Yaskawa INFORM job: DEMO_ROOF_UPPER_0625_3PAINT_16.JBI

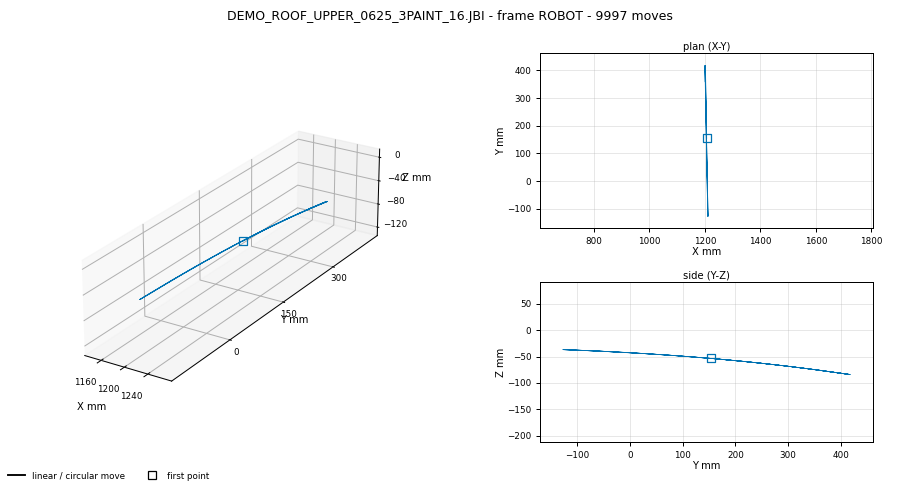
[picture p0: tool path of DEMO_ROOF_UPPER_0625_3PAINT_16.JBI in frame ROBOT, 9997 of 9997 moves have a stored position in this frame; points joined in program order, loops and branches not executed]
/JOB
//NAME DEMO_ROOF_UPPER_0625_3PAINT16
//POS
///NPOS 9997,0,0,0,0,0
///TOOL 0
///USER 0
///POSTYPE ROBOT
///RECTAN
///RCONF 1,0,0,0,0,0,0,0,0,0,0,0,0,0,0,0,0,0,0,0,0,0,0,0
C00000=1206.516,154.392,-53.585,-178.084,6.068,148.520
C00001=1206.512,154.641,-53.607,-178.082,6.070,148.519
C00002=1206.507,154.891,-53.628,-178.079,6.072,148.519
C00003=1206.502,155.139,-53.650,-178.077,6.072,148.518
C00004=1206.498,155.388,-53.670,-178.074,6.074,148.518
C00005=1206.493,155.637,-53.692,-178.071,6.076,148.517
C00006=1206.488,155.887,-53.713,-178.068,6.078,148.517
C00007=1206.483,156.135,-53.735,-178.066,6.078,148.517
C00008=1206.479,156.384,-53.757,-178.063,6.080,148.516
C00009=1206.473,156.633,-53.778,-178.060,6.082,148.516
C00010=1206.470,156.882,-53.799,-178.058,6.083,148.515
C00011=1206.465,157.131,-53.821,-178.056,6.085,148.515
C00012=1206.460,157.380,-53.842,-178.053,6.086,148.515
C00013=1206.456,157.630,-53.864,-178.050,6.087,148.514
C00014=1206.450,157.879,-53.885,-178.048,6.089,148.514
C00015=1206.445,158.127,-53.906,-178.045,6.091,148.513
C00016=1206.441,158.377,-53.928,-178.043,6.092,148.513
C00017=1206.436,158.625,-53.950,-178.040,6.093,148.512
C00018=1206.432,158.894,-53.973,-178.037,6.095,148.512
C00019=1206.426,159.164,-53.996,-178.034,6.097,148.511
C00020=1206.421,159.433,-54.019,-178.031,6.098,148.511
C00021=1206.416,159.702,-54.043,-178.028,6.100,148.510
C00022=1206.411,159.950,-54.065,-178.026,6.101,148.510
C00023=1206.407,160.200,-54.086,-178.023,6.102,148.509
C00024=1206.402,160.449,-54.108,-178.021,6.104,148.509
C00025=1206.397,160.698,-54.130,-178.018,6.106,148.509
C00026=1206.393,160.947,-54.152,-178.016,6.107,148.508
C00027=1206.388,161.196,-54.172,-178.013,6.109,148.508
C00028=1206.383,161.444,-54.194,-178.010,6.110,148.507
C00029=1206.379,161.694,-54.216,-178.008,6.111,148.507
C00030=1206.374,161.942,-54.237,-178.005,6.113,148.507
C00031=1206.370,162.192,-54.259,-178.002,6.115,148.506
C00032=1206.365,162.440,-54.281,-178.000,6.116,148.506
C00033=1206.360,162.690,-54.302,-177.997,6.117,148.505
C00034=1206.355,162.939,-54.325,-177.995,6.119,148.505
C00035=1206.350,163.188,-54.346,-177.992,6.121,148.505
C00036=1206.346,163.437,-54.368,-177.990,6.122,148.504
C00037=1206.341,163.686,-54.390,-177.987,6.123,148.504
C00038=1206.337,163.935,-54.412,-177.984,6.125,148.503
C00039=1206.332,164.184,-54.434,-177.981,6.127,148.503
C00040=1206.327,164.433,-54.456,-177.979,6.128,148.502
C00041=1206.323,164.682,-54.478,-177.977,6.130,148.502
C00042=1206.318,164.931,-54.499,-177.974,6.131,148.502
C00043=1206.314,165.180,-54.521,-177.971,6.133,148.501
C00044=1206.309,165.429,-54.543,-177.969,6.134,148.501
C00045=1206.304,165.678,-54.565,-177.966,6.136,148.500
C00046=1206.300,165.927,-54.587,-177.963,6.137,148.500
C00047=1206.295,166.176,-54.609,-177.961,6.139,148.500
C00048=1206.290,166.425,-54.631,-177.959,6.140,148.499
C00049=1206.285,166.674,-54.653,-177.955,6.142,148.499
C00050=1206.281,166.923,-54.675,-177.953,6.143,148.498
C00051=1206.276,167.171,-54.696,-177.950,6.145,148.498
C00052=1206.271,167.421,-54.718,-177.948,6.146,148.498
C00053=1206.267,167.669,-54.740,-177.945,6.148,148.497
C00054=1206.262,167.919,-54.762,-177.943,6.150,148.497
C00055=1206.257,168.168,-54.784,-177.939,6.151,148.496
C00056=1206.252,168.417,-54.807,-177.937,6.152,148.496
C00057=1206.248,168.666,-54.828,-177.935,6.154,148.495
C00058=1206.244,168.914,-54.851,-177.932,6.156,148.495
C00059=1206.239,169.163,-54.873,-177.929,6.158,148.495
C00060=1206.234,169.413,-54.895,-177.927,6.159,148.494
C00061=1206.229,169.661,-54.917,-177.924,6.160,148.494
C00062=1206.225,169.911,-54.939,-177.921,6.162,148.493
C00063=1206.220,170.160,-54.961,-177.919,6.164,148.493
C00064=1206.215,170.408,-54.984,-177.916,6.166,148.493
C00065=1206.211,170.658,-55.006,-177.914,6.166,148.492
C00066=1206.206,170.906,-55.028,-177.911,6.168,148.492
C00067=1206.202,171.156,-55.050,-177.909,6.170,148.492
C00068=1206.196,171.405,-55.072,-177.906,6.172,148.491
C00069=1206.192,171.653,-55.095,-177.903,6.173,148.491
C00070=1206.187,171.902,-55.117,-177.901,6.174,148.490
C00071=1206.183,172.151,-55.139,-177.898,6.176,148.490
C00072=1206.178,172.401,-55.161,-177.895,6.178,148.489
C00073=1206.173,172.649,-55.184,-177.893,6.180,148.489
C00074=1206.169,172.898,-55.206,-177.891,6.181,148.489
C00075=1206.163,173.147,-55.228,-177.888,6.182,148.488
C00076=1206.159,173.396,-55.251,-177.885,6.184,148.488
C00077=1206.155,173.645,-55.272,-177.882,6.186,148.487
C00078=1206.150,173.894,-55.295,-177.880,6.188,148.487
C00079=1206.146,174.143,-55.318,-177.877,6.189,148.487
C00080=1206.141,174.392,-55.340,-177.875,6.190,148.486
C00081=1206.136,174.641,-55.362,-177.872,6.192,148.486
C00082=1206.132,174.890,-55.385,-177.869,6.194,148.486
C00083=1206.127,175.139,-55.407,-177.866,6.196,148.485
C00084=1206.122,175.388,-55.430,-177.864,6.197,148.485
C00085=1206.117,175.636,-55.452,-177.862,6.198,148.484
C00086=1206.112,175.886,-55.474,-177.859,6.200,148.484
C00087=1206.108,176.135,-55.497,-177.856,6.202,148.484
C00088=1206.104,176.383,-55.519,-177.854,6.204,148.483
C00089=1206.099,176.632,-55.542,-177.851,6.205,148.483
C00090=1206.095,176.882,-55.564,-177.849,6.207,148.482
C00091=1206.089,177.130,-55.587,-177.846,6.208,148.482
C00092=1206.085,177.379,-55.609,-177.843,6.210,148.482
C00093=1206.081,177.628,-55.632,-177.840,6.212,148.481
C00094=1206.075,177.877,-55.654,-177.838,6.213,148.481
C00095=1206.071,178.126,-55.677,-177.836,6.214,148.480
C00096=1206.066,178.375,-55.700,-177.833,6.216,148.480
C00097=1206.062,178.623,-55.722,-177.830,6.218,148.480
C00098=1206.057,178.873,-55.745,-177.828,6.220,148.479
C00099=1206.053,179.122,-55.767,-177.825,6.222,148.479
C00100=1206.047,179.371,-55.790,-177.823,6.223,148.479
C00101=1206.043,179.620,-55.813,-177.820,6.224,148.478
C00102=1206.039,179.869,-55.836,-177.817,6.226,148.478
C00103=1206.034,180.118,-55.858,-177.814,6.228,148.477
C00104=1206.029,180.366,-55.881,-177.812,6.230,148.477
C00105=1206.025,180.616,-55.903,-177.809,6.231,148.477
C00106=1206.020,180.865,-55.926,-177.806,6.233,148.476
C00107=1206.016,181.113,-55.949,-177.804,6.234,148.476
C00108=1206.011,181.362,-55.971,-177.802,6.236,148.476
C00109=1206.007,181.611,-55.994,-177.799,6.238,148.475
C00110=1206.002,181.860,-56.017,-177.796,6.240,148.475
C00111=1205.996,182.109,-56.040,-177.794,6.241,148.474
C00112=1205.992,182.358,-56.063,-177.791,6.243,148.474
C00113=1205.988,182.607,-56.086,-177.789,6.244,148.474
C00114=1205.984,182.855,-56.109,-177.786,6.246,148.473
C00115=1205.978,183.104,-56.131,-177.784,6.248,148.473
C00116=1205.973,183.353,-56.154,-177.780,6.249,148.472
C00117=1205.969,183.602,-56.177,-177.778,6.251,148.472
C00118=1205.964,183.852,-56.200,-177.775,6.253,148.472
C00119=1205.960,184.101,-56.222,-177.772,6.255,148.471
C00120=1205.955,184.349,-56.245,-177.770,6.256,148.471
C00121=1205.950,184.598,-56.269,-177.768,6.258,148.471
C00122=1205.946,184.867,-56.293,-177.765,6.259,148.470
C00123=1205.941,185.137,-56.318,-177.762,6.262,148.470
C00124=1205.935,185.407,-56.343,-177.759,6.264,148.470
C00125=1205.931,185.676,-56.368,-177.756,6.265,148.469
C00126=1205.926,185.925,-56.391,-177.753,6.267,148.469
C00127=1205.921,186.174,-56.414,-177.751,6.269,148.468
C00128=1205.917,186.423,-56.437,-177.749,6.270,148.468
C00129=1205.913,186.672,-56.461,-177.746,6.272,148.468
C00130=1205.907,186.920,-56.484,-177.743,6.274,148.467
C00131=1205.903,187.170,-56.506,-177.741,6.275,148.467
C00132=1205.898,187.419,-56.529,-177.738,6.277,148.467
C00133=1205.894,187.668,-56.552,-177.735,6.279,148.466
C00134=1205.889,187.917,-56.576,-177.733,6.281,148.466
C00135=1205.885,188.166,-56.598,-177.730,6.283,148.465
C00136=1205.880,188.414,-56.621,-177.727,6.284,148.465
C00137=1205.875,188.663,-56.645,-177.725,6.285,148.465
C00138=1205.870,188.912,-56.668,-177.723,6.287,148.464
C00139=1205.866,189.161,-56.691,-177.720,6.289,148.464
C00140=1205.862,189.410,-56.714,-177.717,6.291,148.464
C00141=1205.857,189.659,-56.738,-177.715,6.293,148.463
C00142=1205.852,189.908,-56.761,-177.712,6.295,148.463
C00143=1205.847,190.157,-56.784,-177.709,6.296,148.463
C00144=1205.844,190.406,-56.807,-177.707,6.298,148.462
C00145=1205.838,190.654,-56.830,-177.704,6.300,148.462
C00146=1205.834,190.903,-56.854,-177.701,6.302,148.462
C00147=1205.829,191.152,-56.877,-177.699,6.303,148.461
C00148=1205.824,191.401,-56.900,-177.697,6.305,148.461
C00149=1205.820,191.649,-56.924,-177.694,6.306,148.460
C00150=1205.816,191.898,-56.947,-177.691,6.308,148.460
C00151=1205.811,192.147,-56.970,-177.689,6.310,148.460
C00152=1205.806,192.396,-56.994,-177.686,6.312,148.459
C00153=1205.802,192.645,-57.017,-177.683,6.314,148.459
C00154=1205.797,192.894,-57.040,-177.681,6.316,148.459
C00155=1205.792,193.143,-57.064,-177.678,6.317,148.458
C00156=1205.788,193.392,-57.088,-177.675,6.319,148.458
C00157=1205.783,193.641,-57.111,-177.673,6.321,148.458
C00158=1205.778,193.890,-57.135,-177.670,6.323,148.457
C00159=1205.774,194.139,-57.157,-177.667,6.325,148.457
C00160=1205.769,194.387,-57.180,-177.665,6.326,148.457
C00161=1205.765,194.635,-57.204,-177.663,6.327,148.456
C00162=1205.760,194.884,-57.228,-177.660,6.329,148.456
C00163=1205.755,195.133,-57.251,-177.657,6.331,148.456
C00164=1205.751,195.382,-57.275,-177.655,6.333,148.455
C00165=1205.746,195.631,-57.299,-177.652,6.335,148.455
C00166=1205.742,195.880,-57.322,-177.649,6.337,148.455
C00167=1205.737,196.129,-57.345,-177.647,6.338,148.454
C00168=1205.732,196.378,-57.369,-177.644,6.340,148.454
C00169=1205.728,196.626,-57.393,-177.641,6.342,148.454
C00170=1205.723,196.875,-57.416,-177.639,6.344,148.453
C00171=1205.718,197.124,-57.439,-177.636,6.346,148.453
C00172=1205.714,197.373,-57.464,-177.634,6.347,148.452
C00173=1205.710,197.623,-57.487,-177.631,6.349,148.452
C00174=1205.706,197.871,-57.511,-177.628,6.351,148.452
C00175=1205.701,198.120,-57.535,-177.626,6.353,148.451
C00176=1205.696,198.369,-57.558,-177.623,6.355,148.451
C00177=1205.692,198.617,-57.582,-177.620,6.357,148.451
C00178=1205.687,198.866,-57.606,-177.618,6.358,148.450
C00179=1205.683,199.115,-57.630,-177.615,6.360,148.450
C00180=1205.677,199.364,-57.654,-177.613,6.361,148.450
C00181=1205.672,199.613,-57.677,-177.610,6.363,148.449
C00182=1205.668,199.862,-57.701,-177.608,6.365,148.449
C00183=1205.663,200.111,-57.724,-177.605,6.367,148.449
C00184=1205.659,200.359,-57.748,-177.602,6.369,148.448
C00185=1205.654,200.608,-57.772,-177.600,6.370,148.448
C00186=1205.650,200.857,-57.796,-177.597,6.372,148.448
C00187=1205.645,201.106,-57.819,-177.595,6.374,148.448
C00188=1205.641,201.355,-57.844,-177.592,6.376,148.447
C00189=1205.636,201.604,-57.868,-177.590,6.378,148.447
C00190=1205.632,201.852,-57.892,-177.587,6.380,148.446
C00191=1205.627,202.101,-57.916,-177.584,6.382,148.446
C00192=1205.622,202.350,-57.939,-177.582,6.383,148.446
C00193=1205.618,202.598,-57.963,-177.579,6.385,148.445
C00194=1205.613,202.847,-57.987,-177.576,6.387,148.445
C00195=1205.608,203.096,-58.011,-177.574,6.389,148.445
C00196=1205.604,203.345,-58.036,-177.571,6.391,148.444
C00197=1205.600,203.594,-58.059,-177.568,6.393,148.444
C00198=1205.595,203.843,-58.083,-177.566,6.394,148.444
C00199=1205.591,204.092,-58.106,-177.563,6.396,148.443
C00200=1205.586,204.340,-58.131,-177.560,6.398,148.443
C00201=1205.581,204.589,-58.155,-177.558,6.400,148.443
C00202=1205.576,204.838,-58.179,-177.556,6.402,148.443
C00203=1205.573,205.087,-58.203,-177.553,6.404,148.442
C00204=1205.568,205.335,-58.227,-177.550,6.406,148.442
C00205=1205.563,205.584,-58.252,-177.548,6.408,148.442
C00206=1205.558,205.833,-58.275,-177.545,6.409,148.441
C00207=1205.554,206.081,-58.299,-177.542,6.411,148.441
C00208=1205.550,206.331,-58.324,-177.540,6.413,148.441
C00209=1205.545,206.580,-58.348,-177.537,6.415,148.440
C00210=1205.540,206.828,-58.372,-177.534,6.417,148.440
C00211=1205.536,207.077,-58.396,-177.532,6.419,148.440
C00212=1205.531,207.325,-58.420,-177.529,6.420,148.439
C00213=1205.527,207.575,-58.445,-177.527,6.423,148.439
C00214=1205.522,207.824,-58.468,-177.524,6.424,148.439
C00215=1205.517,208.072,-58.493,-177.522,6.426,148.438
C00216=1205.513,208.321,-58.517,-177.519,6.428,148.438
C00217=1205.508,208.569,-58.541,-177.516,6.430,148.438
C00218=1205.504,208.819,-58.566,-177.514,6.432,148.437
C00219=1205.500,209.067,-58.590,-177.511,6.433,148.437
C00220=1205.494,209.316,-58.615,-177.508,6.436,148.437
C00221=1205.490,209.565,-58.638,-177.505,6.438,148.436
C00222=1205.486,209.814,-58.663,-177.503,6.440,148.436
C00223=1205.481,210.063,-58.687,-177.500,6.442,148.436
C00224=1205.476,210.311,-58.711,-177.498,6.444,148.436
C00225=1205.471,210.560,-58.736,-177.495,6.446,148.435
C00226=1205.467,210.830,-58.762,-177.492,6.447,148.435
C00227=1205.462,211.100,-58.789,-177.490,6.449,148.435
C00228=1205.457,211.371,-58.815,-177.487,6.452,148.434
C00229=1205.452,211.641,-58.842,-177.484,6.454,148.434
C00230=1205.448,211.891,-58.866,-177.481,6.456,148.434
C00231=1205.443,212.139,-58.891,-177.479,6.457,148.433
C00232=1205.438,212.388,-58.915,-177.476,6.459,148.433
C00233=1205.434,212.637,-58.940,-177.473,6.461,148.433
C00234=1205.429,212.886,-58.964,-177.471,6.463,148.432
C00235=1205.424,213.134,-58.989,-177.468,6.465,148.432
C00236=1205.421,213.383,-59.013,-177.466,6.467,148.432
C00237=1205.415,213.632,-59.038,-177.463,6.469,148.432
C00238=1205.411,213.880,-59.063,-177.461,6.471,148.431
C00239=1205.406,214.129,-59.087,-177.457,6.473,148.431
C00240=1205.402,214.378,-59.112,-177.455,6.475,148.431
C00241=1205.397,214.626,-59.137,-177.452,6.477,148.430
C00242=1205.393,214.876,-59.161,-177.450,6.479,148.430
C00243=1205.388,215.124,-59.186,-177.447,6.481,148.430
C00244=1205.384,215.373,-59.210,-177.445,6.483,148.429
C00245=1205.379,215.622,-59.235,-177.442,6.485,148.429
C00246=1205.375,215.870,-59.260,-177.439,6.486,148.429
C00247=1205.370,216.119,-59.284,-177.437,6.488,148.428
C00248=1205.366,216.368,-59.309,-177.434,6.490,148.428
C00249=1205.361,216.616,-59.333,-177.432,6.492,148.428
C00250=1205.356,216.865,-59.358,-177.429,6.494,148.428
C00251=1205.353,217.114,-59.383,-177.427,6.496,148.427
C00252=1205.348,217.362,-59.408,-177.424,6.499,148.427
C00253=1205.343,217.612,-59.433,-177.421,6.500,148.427
C00254=1205.339,217.860,-59.457,-177.418,6.502,148.426
C00255=1205.334,218.109,-59.483,-177.416,6.504,148.426
C00256=1205.329,218.358,-59.507,-177.413,6.506,148.426
C00257=1205.325,218.606,-59.531,-177.411,6.508,148.426
C00258=1205.321,218.855,-59.557,-177.408,6.510,148.425
C00259=1205.316,219.103,-59.581,-177.406,6.512,148.425
C00260=1205.312,219.353,-59.606,-177.403,6.514,148.425
C00261=1205.307,219.601,-59.632,-177.401,6.516,148.424
C00262=1205.303,219.850,-59.656,-177.398,6.518,148.424
C00263=1205.298,220.099,-59.681,-177.395,6.520,148.424
C00264=1205.293,220.347,-59.706,-177.392,6.522,148.424
C00265=1205.289,220.596,-59.731,-177.390,6.524,148.423
C00266=1205.284,220.845,-59.755,-177.387,6.526,148.423
C00267=1205.280,221.094,-59.781,-177.385,6.528,148.423
C00268=1205.275,221.342,-59.806,-177.382,6.530,148.422
C00269=1205.271,221.591,-59.831,-177.380,6.532,148.422
C00270=1205.266,221.839,-59.856,-177.377,6.533,148.422
C00271=1205.262,222.088,-59.881,-177.375,6.536,148.422
C00272=1205.257,222.337,-59.906,-177.372,6.537,148.421
C00273=1205.253,222.585,-59.931,-177.369,6.540,148.421
C00274=1205.248,222.834,-59.956,-177.366,6.542,148.421
C00275=1205.244,223.083,-59.982,-177.364,6.544,148.420
C00276=1205.239,223.332,-60.006,-177.361,6.546,148.420
C00277=1205.235,223.581,-60.032,-177.359,6.548,148.420
C00278=1205.230,223.829,-60.056,-177.356,6.550,148.420
C00279=1205.226,224.078,-60.082,-177.354,6.551,148.419
C00280=1205.221,224.326,-60.106,-177.351,6.554,148.419
C00281=1205.217,224.575,-60.132,-177.348,6.556,148.419
C00282=1205.212,224.824,-60.157,-177.346,6.558,148.419
C00283=1205.207,225.073,-60.183,-177.343,6.560,148.418
C00284=1205.203,225.321,-60.207,-177.341,6.562,148.418
C00285=1205.199,225.570,-60.232,-177.338,6.564,148.418
C00286=1205.194,225.819,-60.258,-177.335,6.566,148.417
C00287=1205.189,226.068,-60.283,-177.333,6.568,148.417
C00288=1205.185,226.316,-60.309,-177.330,6.569,148.417
C00289=1205.180,226.564,-60.334,-177.328,6.572,148.417
C00290=1205.176,226.814,-60.359,-177.325,6.574,148.416
C00291=1205.171,227.062,-60.384,-177.322,6.576,148.416
C00292=1205.167,227.311,-60.410,-177.320,6.578,148.416
C00293=1205.163,227.559,-60.435,-177.317,6.580,148.416
C00294=1205.158,227.808,-60.460,-177.315,6.582,148.415
C00295=1205.154,228.057,-60.486,-177.312,6.584,148.415
C00296=1205.149,228.305,-60.511,-177.310,6.586,148.415
C00297=1205.145,228.554,-60.536,-177.307,6.589,148.415
C00298=1205.140,228.803,-60.562,-177.304,6.591,148.414
C00299=1205.135,229.051,-60.587,-177.302,6.592,148.414
C00300=1205.131,229.300,-60.613,-177.299,6.595,148.414
C00301=1205.126,229.548,-60.638,-177.297,6.596,148.414
C00302=1205.122,229.798,-60.663,-177.294,6.598,148.413
C00303=1205.118,230.046,-60.689,-177.291,6.600,148.413
C00304=1205.113,230.294,-60.715,-177.289,6.603,148.413
C00305=1205.109,230.543,-60.740,-177.286,6.605,148.413
C00306=1205.104,230.792,-60.766,-177.283,6.607,148.412
C00307=1205.100,231.040,-60.791,-177.281,6.609,148.412
C00308=1205.095,231.290,-60.817,-177.279,6.611,148.412
C00309=1205.091,231.538,-60.842,-177.276,6.613,148.411
C00310=1205.086,231.787,-60.868,-177.273,6.614,148.411
C00311=1205.082,232.035,-60.893,-177.271,6.617,148.411
C00312=1205.078,232.284,-60.919,-177.268,6.619,148.411
C00313=1205.073,232.532,-60.945,-177.265,6.621,148.410
C00314=1205.068,232.781,-60.971,-177.263,6.623,148.410
C00315=1205.064,233.030,-60.997,-177.261,6.625,148.410
C00316=1205.059,233.278,-61.022,-177.258,6.627,148.410
C00317=1205.054,233.527,-61.048,-177.255,6.630,148.410
C00318=1205.050,233.776,-61.074,-177.253,6.632,148.409
C00319=1205.045,234.024,-61.099,-177.250,6.634,148.409
C00320=1205.041,234.273,-61.125,-177.247,6.636,148.409
C00321=1205.037,234.522,-61.150,-177.245,6.638,148.409
C00322=1205.033,234.770,-61.176,-177.243,6.640,148.408
C00323=1205.027,235.019,-61.202,-177.239,6.642,148.408
C00324=1205.023,235.268,-61.228,-177.237,6.644,148.408
C00325=1205.019,235.516,-61.254,-177.235,6.646,148.407
C00326=1205.014,235.765,-61.279,-177.232,6.648,148.407
C00327=1205.010,236.013,-61.305,-177.230,6.650,148.407
C00328=1205.005,236.262,-61.331,-177.227,6.653,148.407
C00329=1205.000,236.511,-61.357,-177.224,6.655,148.406
C00330=1204.995,236.782,-61.385,-177.222,6.657,148.406
C00331=1204.991,237.054,-61.413,-177.219,6.660,148.406
C00332=1204.986,237.325,-61.442,-177.216,6.661,148.406
C00333=1204.981,237.596,-61.470,-177.213,6.664,148.405
C00334=1204.977,237.845,-61.495,-177.211,6.666,148.405
C00335=1204.972,238.094,-61.522,-177.208,6.668,148.405
C00336=1204.968,238.342,-61.548,-177.205,6.670,148.405
C00337=1204.963,238.590,-61.574,-177.203,6.672,148.405
C00338=1204.959,238.839,-61.599,-177.200,6.675,148.404
C00339=1204.954,239.088,-61.626,-177.197,6.677,148.404
C00340=1204.950,239.337,-61.652,-177.195,6.679,148.404
C00341=1204.946,239.585,-61.678,-177.193,6.681,148.404
C00342=1204.940,239.834,-61.704,-177.190,6.683,148.403
C00343=1204.936,240.083,-61.730,-177.187,6.686,148.403
C00344=1204.932,240.331,-61.756,-177.185,6.687,148.403
C00345=1204.928,240.580,-61.782,-177.182,6.689,148.403
C00346=1204.923,240.829,-61.808,-177.180,6.691,148.403
C00347=1204.919,241.077,-61.834,-177.177,6.693,148.402
C00348=1204.914,241.325,-61.860,-177.175,6.696,148.402
C00349=1204.909,241.574,-61.886,-177.172,6.698,148.402
C00350=1204.905,241.822,-61.913,-177.169,6.700,148.402
C00351=1204.900,242.071,-61.939,-177.167,6.702,148.401
C00352=1204.896,242.320,-61.965,-177.164,6.705,148.401
C00353=1204.892,242.568,-61.992,-177.162,6.707,148.401
C00354=1204.887,242.817,-62.018,-177.159,6.709,148.401
C00355=1204.883,243.066,-62.044,-177.157,6.711,148.400
C00356=1204.879,243.314,-62.070,-177.154,6.713,148.400
C00357=1204.874,243.563,-62.096,-177.151,6.716,148.400
C00358=1204.870,243.811,-62.123,-177.149,6.717,148.400
C00359=1204.865,244.060,-62.149,-177.146,6.720,148.400
C00360=1204.861,244.308,-62.175,-177.144,6.721,148.399
C00361=1204.856,244.557,-62.202,-177.141,6.724,148.399
C00362=1204.852,244.806,-62.228,-177.138,6.726,148.399
C00363=1204.848,245.054,-62.254,-177.136,6.728,148.399
C00364=1204.843,245.303,-62.281,-177.134,6.730,148.399
C00365=1204.839,245.552,-62.307,-177.131,6.733,148.398
C00366=1204.834,245.800,-62.333,-177.128,6.735,148.398
C00367=1204.829,246.048,-62.359,-177.126,6.737,148.398
C00368=1204.825,246.297,-62.386,-177.124,6.739,148.398
C00369=1204.821,246.545,-62.413,-177.120,6.742,148.397
C00370=1204.816,246.794,-62.439,-177.118,6.744,148.397
C00371=1204.812,247.042,-62.465,-177.116,6.746,148.397
C00372=1204.807,247.291,-62.492,-177.113,6.748,148.397
C00373=1204.803,247.540,-62.518,-177.110,6.751,148.397
C00374=1204.798,247.788,-62.545,-177.108,6.753,148.396
C00375=1204.794,248.037,-62.571,-177.106,6.755,148.396
C00376=1204.789,248.285,-62.598,-177.103,6.757,148.396
C00377=1204.785,248.534,-62.625,-177.100,6.759,148.396
C00378=1204.781,248.783,-62.651,-177.098,6.761,148.396
C00379=1204.776,249.031,-62.678,-177.095,6.763,148.395
C00380=1204.772,249.279,-62.705,-177.093,6.766,148.395
C00381=1204.767,249.529,-62.731,-177.090,6.768,148.395
C00382=1204.762,249.777,-62.758,-177.087,6.770,148.395
C00383=1204.758,250.025,-62.784,-177.085,6.772,148.395
C00384=1204.754,250.274,-62.811,-177.083,6.774,148.394
C00385=1204.750,250.523,-62.837,-177.079,6.777,148.394
C00386=1204.745,250.771,-62.864,-177.077,6.779,148.394
C00387=1204.740,251.019,-62.891,-177.075,6.781,148.394
C00388=1204.736,251.268,-62.918,-177.072,6.784,148.394
C00389=1204.732,251.516,-62.945,-177.069,6.786,148.393
C00390=1204.727,251.765,-62.971,-177.067,6.788,148.393
C00391=1204.723,252.013,-62.998,-177.065,6.790,148.393
C00392=1204.718,252.262,-63.025,-177.061,6.793,148.393
C00393=1204.713,252.510,-63.052,-177.059,6.795,148.393
C00394=1204.710,252.759,-63.078,-177.057,6.797,148.392
C00395=1204.705,253.007,-63.105,-177.054,6.800,148.392
C00396=1204.700,253.256,-63.132,-177.051,6.802,148.392
C00397=1204.697,253.505,-63.159,-177.049,6.804,148.392
C00398=1204.692,253.754,-63.186,-177.046,6.806,148.392
C00399=1204.687,254.002,-63.213,-177.044,6.809,148.392
C00400=1204.683,254.251,-63.240,-177.041,6.810,148.391
C00401=1204.679,254.499,-63.266,-177.039,6.813,148.391
C00402=1204.674,254.747,-63.293,-177.036,6.815,148.391
C00403=1204.669,254.996,-63.320,-177.034,6.818,148.391
C00404=1204.665,255.244,-63.347,-177.031,6.819,148.390
C00405=1204.661,255.492,-63.374,-177.028,6.822,148.390
C00406=1204.656,255.741,-63.401,-177.026,6.824,148.390
C00407=1204.652,255.990,-63.428,-177.024,6.826,148.390
C00408=1204.647,256.239,-63.455,-177.020,6.829,148.390
C00409=1204.643,256.487,-63.482,-177.018,6.831,148.390
C00410=1204.639,256.735,-63.509,-177.016,6.833,148.389
C00411=1204.634,256.984,-63.536,-177.013,6.836,148.389
C00412=1204.630,257.232,-63.564,-177.010,6.838,148.389
C00413=1204.625,257.480,-63.591,-177.008,6.840,148.389
C00414=1204.621,257.729,-63.618,-177.005,6.843,148.389
C00415=1204.617,257.978,-63.645,-177.003,6.845,148.389
C00416=1204.613,258.226,-63.672,-177.000,6.847,148.388
C00417=1204.608,258.475,-63.699,-176.998,6.849,148.388
C00418=1204.603,258.723,-63.726,-176.995,6.852,148.388
C00419=1204.599,258.972,-63.753,-176.993,6.854,148.388
C00420=1204.594,259.219,-63.781,-176.990,6.856,148.388
C00421=1204.590,259.469,-63.808,-176.987,6.859,148.387
C00422=1204.586,259.717,-63.835,-176.985,6.861,148.387
C00423=1204.581,259.966,-63.862,-176.982,6.864,148.387
C00424=1204.576,260.214,-63.889,-176.980,6.866,148.387
C00425=1204.572,260.462,-63.917,-176.977,6.868,148.387
C00426=1204.568,260.711,-63.945,-176.975,6.871,148.387
C00427=1204.564,260.959,-63.971,-176.972,6.873,148.386
C00428=1204.559,261.208,-63.998,-176.970,6.875,148.386
C00429=1204.555,261.456,-64.026,-176.967,6.877,148.386
C00430=1204.551,261.705,-64.053,-176.965,6.880,148.386
C00431=1204.546,261.953,-64.080,-176.962,6.881,148.386
C00432=1204.542,262.201,-64.108,-176.959,6.885,148.386
C00433=1204.537,262.450,-64.135,-176.957,6.887,148.386
C00434=1204.533,262.723,-64.166,-176.954,6.889,148.385
C00435=1204.528,262.995,-64.196,-176.951,6.891,148.385
C00436=1204.523,263.268,-64.226,-176.949,6.894,148.385
C00437=1204.517,263.541,-64.256,-176.945,6.897,148.385
C00438=1204.513,263.790,-64.284,-176.943,6.899,148.385
C00439=1204.509,264.038,-64.311,-176.940,6.902,148.384
C00440=1204.504,264.286,-64.338,-176.938,6.904,148.384
C00441=1204.500,264.535,-64.365,-176.936,6.906,148.384
C00442=1204.496,264.783,-64.394,-176.933,6.909,148.384
C00443=1204.491,265.032,-64.421,-176.931,6.911,148.384
C00444=1204.487,265.280,-64.448,-176.928,6.913,148.384
C00445=1204.483,265.529,-64.476,-176.925,6.916,148.383
C00446=1204.479,265.777,-64.504,-176.923,6.918,148.383
C00447=1204.474,266.025,-64.531,-176.920,6.921,148.383
C00448=1204.469,266.274,-64.559,-176.918,6.923,148.383
C00449=1204.465,266.523,-64.587,-176.915,6.925,148.383
C00450=1204.460,266.771,-64.614,-176.912,6.928,148.383
C00451=1204.456,267.020,-64.642,-176.910,6.930,148.383
C00452=1204.452,267.268,-64.670,-176.908,6.932,148.382
C00453=1204.447,267.516,-64.697,-176.905,6.935,148.382
C00454=1204.444,267.765,-64.725,-176.902,6.937,148.382
C00455=1204.438,268.014,-64.752,-176.900,6.940,148.382
C00456=1204.434,268.261,-64.780,-176.898,6.942,148.382
C00457=1204.430,268.510,-64.808,-176.895,6.944,148.382
C00458=1204.425,268.758,-64.835,-176.892,6.947,148.382
C00459=1204.421,269.006,-64.863,-176.890,6.949,148.381
C00460=1204.417,269.255,-64.892,-176.887,6.952,148.381
C00461=1204.412,269.504,-64.919,-176.885,6.954,148.381
C00462=1204.408,269.752,-64.947,-176.882,6.957,148.381
C00463=1204.404,270.000,-64.975,-176.879,6.959,148.381
C00464=1204.399,270.249,-65.002,-176.877,6.961,148.381
C00465=1204.395,270.498,-65.031,-176.874,6.964,148.380
C00466=1204.390,270.745,-65.058,-176.872,6.966,148.380
C00467=1204.386,270.993,-65.086,-176.869,6.969,148.380
C00468=1204.382,271.242,-65.114,-176.867,6.971,148.380
C00469=1204.377,271.491,-65.142,-176.865,6.973,148.380
C00470=1204.373,271.739,-65.170,-176.862,6.976,148.380
C00471=1204.369,271.987,-65.198,-176.859,6.978,148.380
C00472=1204.363,272.236,-65.226,-176.857,6.981,148.380
C00473=1204.360,272.485,-65.254,-176.854,6.983,148.379
C00474=1204.355,272.732,-65.281,-176.851,6.986,148.379
C00475=1204.351,272.981,-65.310,-176.849,6.988,148.379
C00476=1204.346,273.229,-65.338,-176.847,6.990,148.379
C00477=1204.343,273.478,-65.366,-176.844,6.993,148.379
C00478=1204.337,273.727,-65.394,-176.842,6.995,148.379
C00479=1204.334,273.975,-65.422,-176.839,6.998,148.379
C00480=1204.329,274.223,-65.450,-176.836,7.000,148.378
C00481=1204.325,274.472,-65.478,-176.834,7.003,148.378
C00482=1204.320,274.720,-65.506,-176.831,7.005,148.378
C00483=1204.317,274.968,-65.534,-176.829,7.007,148.378
C00484=1204.312,275.217,-65.563,-176.826,7.010,148.378
C00485=1204.307,275.464,-65.591,-176.824,7.012,148.378
C00486=1204.303,275.713,-65.619,-176.821,7.015,148.378
C00487=1204.298,275.961,-65.647,-176.819,7.017,148.378
C00488=1204.295,276.210,-65.675,-176.816,7.020,148.378
C00489=1204.290,276.459,-65.704,-176.814,7.022,148.377
C00490=1204.286,276.706,-65.732,-176.811,7.025,148.377
C00491=1204.281,276.955,-65.760,-176.809,7.027,148.377
C00492=1204.277,277.203,-65.788,-176.806,7.030,148.377
C00493=1204.272,277.452,-65.817,-176.803,7.032,148.377
C00494=1204.268,277.700,-65.845,-176.801,7.034,148.377
C00495=1204.264,277.949,-65.873,-176.798,7.037,148.377
C00496=1204.259,278.197,-65.901,-176.796,7.039,148.377
C00497=1204.255,278.446,-65.930,-176.793,7.042,148.376
C00498=1204.250,278.694,-65.958,-176.791,7.044,148.376
C00499=1204.246,278.942,-65.987,-176.788,7.047,148.376
C00500=1204.242,279.190,-66.015,-176.786,7.049,148.376
C00501=1204.237,279.439,-66.044,-176.783,7.052,148.376
C00502=1204.234,279.687,-66.072,-176.781,7.054,148.376
C00503=1204.229,279.935,-66.100,-176.778,7.057,148.376
C00504=1204.225,280.184,-66.128,-176.775,7.059,148.376
C00505=1204.220,280.431,-66.157,-176.773,7.062,148.376
C00506=1204.216,280.680,-66.186,-176.771,7.064,148.375
C00507=1204.212,280.929,-66.214,-176.768,7.067,148.375
C00508=1204.207,281.177,-66.243,-176.765,7.069,148.375
C00509=1204.203,281.425,-66.272,-176.763,7.072,148.375
C00510=1204.198,281.673,-66.300,-176.761,7.074,148.375
C00511=1204.194,281.922,-66.328,-176.758,7.077,148.375
C00512=1204.190,282.171,-66.357,-176.755,7.079,148.375
C00513=1204.185,282.418,-66.386,-176.753,7.082,148.375
C00514=1204.181,282.667,-66.414,-176.750,7.085,148.375
C00515=1204.177,282.916,-66.443,-176.748,7.088,148.375
C00516=1204.172,283.163,-66.472,-176.746,7.090,148.375
C00517=1204.168,283.412,-66.500,-176.742,7.092,148.374
C00518=1204.163,283.660,-66.528,-176.740,7.095,148.374
C00519=1204.159,283.908,-66.558,-176.738,7.098,148.374
C00520=1204.155,284.157,-66.586,-176.735,7.100,148.374
C00521=1204.150,284.405,-66.614,-176.733,7.103,148.374
C00522=1204.146,284.653,-66.644,-176.730,7.105,148.374
C00523=1204.142,284.902,-66.672,-176.727,7.108,148.374
C00524=1204.138,285.150,-66.701,-176.725,7.110,148.374
C00525=1204.133,285.398,-66.730,-176.723,7.113,148.374
C00526=1204.130,285.646,-66.759,-176.720,7.115,148.374
C00527=1204.125,285.895,-66.787,-176.717,7.118,148.373
C00528=1204.120,286.143,-66.816,-176.715,7.120,148.373
C00529=1204.116,286.392,-66.845,-176.712,7.123,148.373
C00530=1204.112,286.640,-66.874,-176.710,7.125,148.373
C00531=1204.107,286.888,-66.902,-176.708,7.128,148.373
C00532=1204.103,287.136,-66.932,-176.705,7.130,148.373
C00533=1204.099,287.385,-66.961,-176.702,7.133,148.373
C00534=1204.094,287.633,-66.990,-176.700,7.135,148.373
C00535=1204.090,287.881,-67.018,-176.697,7.138,148.373
C00536=1204.086,288.129,-67.047,-176.695,7.141,148.373
C00537=1204.081,288.378,-67.076,-176.693,7.144,148.373
C00538=1204.077,288.652,-67.108,-176.689,7.146,148.372
C00539=1204.072,288.926,-67.140,-176.687,7.149,148.372
C00540=1204.067,289.201,-67.172,-176.684,7.152,148.372
C00541=1204.062,289.475,-67.205,-176.682,7.154,148.372
C00542=1204.058,289.724,-67.233,-176.679,7.157,148.372
C00543=1204.053,289.972,-67.263,-176.676,7.160,148.372
C00544=1204.049,290.219,-67.291,-176.674,7.162,148.372
C00545=1204.045,290.468,-67.320,-176.671,7.165,148.372
C00546=1204.041,290.716,-67.350,-176.669,7.168,148.372
C00547=1204.037,290.965,-67.379,-176.666,7.171,148.372
C00548=1204.032,291.214,-67.408,-176.664,7.173,148.372
C00549=1204.027,291.461,-67.437,-176.661,7.176,148.372
C00550=1204.023,291.709,-67.466,-176.659,7.178,148.371
C00551=1204.019,291.958,-67.496,-176.656,7.181,148.371
C00552=1204.014,292.207,-67.524,-176.654,7.183,148.371
C00553=1204.010,292.455,-67.554,-176.652,7.186,148.371
C00554=1204.005,292.702,-67.583,-176.649,7.189,148.371
C00555=1204.002,292.950,-67.612,-176.647,7.191,148.371
C00556=1203.998,293.199,-67.641,-176.644,7.194,148.371
C00557=1203.994,293.447,-67.671,-176.642,7.196,148.371
C00558=1203.989,293.696,-67.700,-176.639,7.199,148.371
C00559=1203.985,293.944,-67.729,-176.637,7.201,148.371
C00560=1203.981,294.192,-67.758,-176.634,7.204,148.371
C00561=1203.976,294.440,-67.787,-176.632,7.207,148.371
C00562=1203.972,294.688,-67.817,-176.629,7.210,148.371
C00563=1203.968,294.936,-67.846,-176.626,7.213,148.371
C00564=1203.963,295.185,-67.876,-176.624,7.215,148.371
C00565=1203.959,295.433,-67.905,-176.622,7.218,148.371
C00566=1203.954,295.682,-67.935,-176.619,7.220,148.371
C00567=1203.950,295.930,-67.965,-176.617,7.223,148.371
C00568=1203.946,296.178,-67.994,-176.615,7.225,148.371
C00569=1203.941,296.426,-68.023,-176.612,7.228,148.371
C00570=1203.937,296.674,-68.053,-176.609,7.231,148.371
C00571=1203.933,296.922,-68.082,-176.607,7.233,148.370
C00572=1203.929,297.170,-68.112,-176.604,7.236,148.370
C00573=1203.924,297.419,-68.141,-176.602,7.238,148.370
C00574=1203.920,297.667,-68.171,-176.599,7.241,148.370
C00575=1203.916,297.915,-68.200,-176.597,7.244,148.370
C00576=1203.912,298.163,-68.230,-176.594,7.247,148.370
C00577=1203.908,298.412,-68.259,-176.592,7.250,148.370
C00578=1203.903,298.660,-68.289,-176.589,7.252,148.370
C00579=1203.899,298.909,-68.318,-176.587,7.255,148.370
C00580=1203.894,299.157,-68.348,-176.585,7.257,148.370
C00581=1203.890,299.405,-68.377,-176.582,7.260,148.370
C00582=1203.886,299.653,-68.408,-176.580,7.262,148.370
C00583=1203.882,299.900,-68.437,-176.577,7.265,148.370
C00584=1203.877,300.149,-68.467,-176.574,7.268,148.370
C00585=1203.873,300.397,-68.496,-176.572,7.270,148.370
C00586=1203.868,300.645,-68.526,-176.570,7.273,148.370
C00587=1203.864,300.894,-68.555,-176.567,7.276,148.370
C00588=1203.860,301.141,-68.585,-176.565,7.279,148.370
C00589=1203.855,301.390,-68.615,-176.562,7.282,148.370
C00590=1203.851,301.638,-68.645,-176.560,7.284,148.370
C00591=1203.847,301.886,-68.674,-176.557,7.287,148.370
C00592=1203.843,302.134,-68.704,-176.555,7.289,148.369
C00593=1203.838,302.383,-68.734,-176.552,7.292,148.369
C00594=1203.834,302.631,-68.764,-176.550,7.295,148.369
C00595=1203.830,302.879,-68.794,-176.548,7.297,148.369
C00596=1203.825,303.127,-68.824,-176.545,7.300,148.369
C00597=1203.821,303.375,-68.854,-176.543,7.303,148.369
C00598=1203.817,303.624,-68.883,-176.540,7.306,148.369
C00599=1203.813,303.871,-68.913,-176.537,7.309,148.369
C00600=1203.809,304.121,-68.944,-176.536,7.311,148.369
C00601=1203.805,304.368,-68.974,-176.533,7.314,148.369
C00602=1203.801,304.617,-69.003,-176.531,7.316,148.369
C00603=1203.796,304.865,-69.033,-176.528,7.319,148.369
C00604=1203.792,305.113,-69.063,-176.526,7.322,148.369
C00605=1203.787,305.361,-69.093,-176.523,7.325,148.369
C00606=1203.783,305.609,-69.124,-176.521,7.328,148.369
C00607=1203.779,305.857,-69.153,-176.518,7.331,148.369
C00608=1203.774,306.105,-69.184,-176.516,7.333,148.369
C00609=1203.770,306.354,-69.213,-176.513,7.336,148.369
C00610=1203.766,306.601,-69.243,-176.511,7.338,148.369
C00611=1203.761,306.850,-69.273,-176.508,7.341,148.369
C00612=1203.757,307.097,-69.304,-176.506,7.344,148.369
C00613=1203.752,307.346,-69.334,-176.504,7.347,148.369
C00614=1203.749,307.594,-69.364,-176.501,7.350,148.369
C00615=1203.744,307.843,-69.394,-176.499,7.352,148.369
C00616=1203.740,308.091,-69.424,-176.497,7.355,148.369
C00617=1203.735,308.339,-69.455,-176.494,7.358,148.369
C00618=1203.732,308.587,-69.485,-176.492,7.360,148.369
C00619=1203.727,308.835,-69.514,-176.489,7.363,148.369
C00620=1203.723,309.083,-69.545,-176.486,7.366,148.369
C00621=1203.719,309.331,-69.575,-176.485,7.369,148.369
C00622=1203.715,309.580,-69.605,-176.482,7.372,148.369
C00623=1203.711,309.828,-69.636,-176.480,7.374,148.369
C00624=1203.706,310.076,-69.666,-176.477,7.377,148.369
C00625=1203.702,310.324,-69.696,-176.474,7.380,148.369
C00626=1203.697,310.572,-69.727,-176.472,7.382,148.369
C00627=1203.693,310.820,-69.757,-176.470,7.385,148.369
C00628=1203.689,311.068,-69.787,-176.467,7.388,148.369
C00629=1203.685,311.317,-69.818,-176.465,7.391,148.369
C00630=1203.681,311.564,-69.848,-176.463,7.394,148.369
C00631=1203.676,311.812,-69.879,-176.460,7.397,148.369
C00632=1203.672,312.061,-69.908,-176.458,7.399,148.369
C00633=1203.667,312.308,-69.939,-176.455,7.402,148.369
C00634=1203.664,312.557,-69.970,-176.453,7.404,148.369
C00635=1203.659,312.805,-70.000,-176.451,7.407,148.369
C00636=1203.655,313.053,-70.031,-176.448,7.410,148.369
C00637=1203.651,313.301,-70.061,-176.446,7.413,148.369
C00638=1203.646,313.549,-70.091,-176.443,7.416,148.369
C00639=1203.642,313.798,-70.123,-176.441,7.419,148.369
C00640=1203.638,314.045,-70.153,-176.439,7.421,148.369
C00641=1203.633,314.293,-70.183,-176.436,7.424,148.369
C00642=1203.628,314.570,-70.217,-176.434,7.427,148.369
C00643=1203.624,314.846,-70.252,-176.431,7.430,148.369
C00644=1203.619,315.122,-70.286,-176.429,7.434,148.370
C00645=1203.614,315.398,-70.320,-176.426,7.437,148.370
C00646=1203.610,315.646,-70.350,-176.423,7.440,148.370
C00647=1203.606,315.895,-70.381,-176.421,7.442,148.370
C00648=1203.602,316.143,-70.412,-176.418,7.445,148.370
C00649=1203.598,316.390,-70.442,-176.416,7.448,148.370
C00650=1203.593,316.638,-70.473,-176.414,7.450,148.370
C00651=1203.589,316.887,-70.504,-176.411,7.454,148.370
C00652=1203.585,317.135,-70.534,-176.409,7.457,148.370
C00653=1203.581,317.382,-70.565,-176.407,7.459,148.370
C00654=1203.577,317.631,-70.596,-176.404,7.462,148.370
C00655=1203.572,317.879,-70.626,-176.402,7.465,148.370
C00656=1203.568,318.127,-70.657,-176.400,7.468,148.370
C00657=1203.564,318.375,-70.688,-176.397,7.471,148.370
C00658=1203.560,318.623,-70.719,-176.395,7.474,148.370
C00659=1203.555,318.871,-70.749,-176.393,7.476,148.370
C00660=1203.551,319.119,-70.781,-176.390,7.479,148.370
C00661=1203.548,319.367,-70.811,-176.388,7.482,148.370
C00662=1203.543,319.615,-70.842,-176.386,7.485,148.370
C00663=1203.539,319.864,-70.873,-176.383,7.488,148.370
C00664=1203.534,320.112,-70.904,-176.381,7.491,148.370
C00665=1203.530,320.360,-70.935,-176.379,7.493,148.370
C00666=1203.526,320.608,-70.966,-176.376,7.496,148.370
C00667=1203.522,320.855,-70.997,-176.374,7.499,148.370
C00668=1203.517,321.103,-71.028,-176.372,7.502,148.371
C00669=1203.513,321.352,-71.059,-176.369,7.505,148.371
C00670=1203.509,321.600,-71.089,-176.367,7.508,148.371
C00671=1203.505,321.848,-71.121,-176.365,7.510,148.371
C00672=1203.501,322.096,-71.152,-176.362,7.513,148.371
C00673=1203.496,322.344,-71.183,-176.360,7.516,148.371
C00674=1203.493,322.592,-71.213,-176.358,7.519,148.371
C00675=1203.488,322.839,-71.245,-176.355,7.522,148.371
C00676=1203.484,323.088,-71.276,-176.354,7.525,148.371
C00677=1203.480,323.336,-71.307,-176.351,7.528,148.371
C00678=1203.475,323.583,-71.338,-176.348,7.531,148.371
C00679=1203.471,323.832,-71.369,-176.347,7.533,148.371
C00680=1203.467,324.080,-71.400,-176.344,7.536,148.371
C00681=1203.463,324.328,-71.432,-176.342,7.539,148.371
C00682=1203.458,324.576,-71.463,-176.339,7.542,148.371
C00683=1203.455,324.824,-71.495,-176.337,7.545,148.372
C00684=1203.450,325.072,-71.525,-176.335,7.548,148.372
C00685=1203.446,325.320,-71.556,-176.332,7.550,148.372
C00686=1203.442,325.568,-71.588,-176.330,7.554,148.372
C00687=1203.437,325.816,-71.619,-176.328,7.557,148.372
C00688=1203.433,326.064,-71.651,-176.326,7.559,148.372
C00689=1203.429,326.312,-71.681,-176.323,7.562,148.372
C00690=1203.425,326.560,-71.713,-176.321,7.565,148.372
C00691=1203.421,326.808,-71.744,-176.319,7.568,148.372
C00692=1203.417,327.056,-71.776,-176.317,7.571,148.372
C00693=1203.412,327.304,-71.806,-176.314,7.574,148.372
C00694=1203.409,327.552,-71.838,-176.312,7.577,148.373
C00695=1203.404,327.800,-71.869,-176.310,7.580,148.373
C00696=1203.400,328.048,-71.901,-176.307,7.583,148.373
C00697=1203.396,328.296,-71.932,-176.305,7.585,148.373
C00698=1203.392,328.544,-71.964,-176.303,7.588,148.373
C00699=1203.387,328.792,-71.994,-176.300,7.592,148.373
C00700=1203.383,329.040,-72.027,-176.299,7.594,148.373
C00701=1203.379,329.288,-72.058,-176.296,7.597,148.373
C00702=1203.375,329.536,-72.089,-176.294,7.600,148.373
C00703=1203.370,329.784,-72.121,-176.292,7.603,148.373
C00704=1203.367,330.032,-72.153,-176.289,7.606,148.373
C00705=1203.362,330.280,-72.183,-176.287,7.609,148.374
C00706=1203.358,330.528,-72.215,-176.285,7.611,148.374
C00707=1203.354,330.776,-72.248,-176.283,7.615,148.374
C00708=1203.349,331.024,-72.278,-176.280,7.618,148.374
C00709=1203.345,331.272,-72.310,-176.279,7.620,148.374
C00710=1203.341,331.519,-72.342,-176.276,7.623,148.374
C00711=1203.337,331.768,-72.373,-176.274,7.627,148.374
C00712=1203.333,332.015,-72.404,-176.272,7.629,148.374
C00713=1203.328,332.264,-72.437,-176.269,7.632,148.374
C00714=1203.324,332.511,-72.468,-176.267,7.636,148.375
C00715=1203.320,332.760,-72.499,-176.265,7.638,148.375
C00716=1203.316,333.008,-72.531,-176.263,7.641,148.375
C00717=1203.311,333.255,-72.563,-176.261,7.644,148.375
C00718=1203.308,333.503,-72.595,-176.258,7.647,148.375
C00719=1203.303,333.751,-72.627,-176.256,7.650,148.375
C00720=1203.300,333.999,-72.659,-176.253,7.653,148.375
C00721=1203.295,334.248,-72.690,-176.252,7.656,148.375
C00722=1203.291,334.495,-72.722,-176.250,7.659,148.376
C00723=1203.287,334.743,-72.754,-176.247,7.662,148.376
C00724=1203.283,334.991,-72.785,-176.245,7.664,148.376
C00725=1203.278,335.239,-72.818,-176.243,7.668,148.376
C00726=1203.274,335.487,-72.849,-176.241,7.671,148.376
C00727=1203.270,335.734,-72.881,-176.239,7.673,148.376
C00728=1203.266,335.983,-72.913,-176.236,7.677,148.376
C00729=1203.262,336.231,-72.945,-176.234,7.680,148.377
C00730=1203.258,336.478,-72.977,-176.232,7.682,148.377
C00731=1203.253,336.726,-73.009,-176.230,7.686,148.377
C00732=1203.249,336.974,-73.041,-176.228,7.689,148.377
C00733=1203.245,337.222,-73.072,-176.226,7.691,148.377
C00734=1203.241,337.470,-73.105,-176.223,7.694,148.377
C00735=1203.237,337.718,-73.137,-176.221,7.698,148.377
C00736=1203.232,337.966,-73.169,-176.219,7.700,148.378
C00737=1203.228,338.214,-73.201,-176.217,7.703,148.378
C00738=1203.225,338.462,-73.232,-176.215,7.707,148.378
C00739=1203.219,338.709,-73.265,-176.213,7.709,148.378
C00740=1203.216,338.957,-73.296,-176.211,7.712,148.378
C00741=1203.211,339.206,-73.329,-176.208,7.716,148.378
C00742=1203.208,339.454,-73.361,-176.206,7.718,148.378
C00743=1203.203,339.701,-73.392,-176.204,7.721,148.379
C00744=1203.199,339.950,-73.425,-176.202,7.725,148.379
C00745=1203.195,340.197,-73.457,-176.200,7.727,148.379
C00746=1203.190,340.475,-73.493,-176.197,7.731,148.379
C00747=1203.186,340.754,-73.529,-176.195,7.734,148.379
C00748=1203.181,341.032,-73.565,-176.193,7.738,148.380
C00749=1203.177,341.310,-73.601,-176.190,7.741,148.380
C00750=1203.172,341.558,-73.634,-176.188,7.744,148.380
C00751=1203.167,341.806,-73.666,-176.186,7.747,148.380
C00752=1203.164,342.054,-73.698,-176.184,7.750,148.380
C00753=1203.159,342.302,-73.730,-176.182,7.754,148.381
C00754=1203.156,342.550,-73.763,-176.180,7.756,148.381
C00755=1203.151,342.797,-73.795,-176.178,7.759,148.381
C00756=1203.147,343.046,-73.827,-176.176,7.762,148.381
C00757=1203.143,343.294,-73.859,-176.174,7.765,148.381
C00758=1203.139,343.541,-73.892,-176.172,7.768,148.381
C00759=1203.134,343.789,-73.924,-176.170,7.771,148.382
C00760=1203.130,344.037,-73.956,-176.168,7.774,148.382
C00761=1203.126,344.285,-73.989,-176.165,7.778,148.382
C00762=1203.122,344.533,-74.021,-176.164,7.780,148.382
C00763=1203.118,344.781,-74.053,-176.162,7.783,148.382
C00764=1203.113,345.028,-74.086,-176.159,7.787,148.383
C00765=1203.110,345.276,-74.118,-176.158,7.789,148.383
C00766=1203.106,345.524,-74.151,-176.155,7.793,148.383
C00767=1203.101,345.772,-74.183,-176.153,7.796,148.383
C00768=1203.097,346.020,-74.215,-176.152,7.798,148.383
C00769=1203.093,346.267,-74.248,-176.149,7.802,148.384
C00770=1203.088,346.516,-74.280,-176.147,7.805,148.384
C00771=1203.085,346.763,-74.313,-176.146,7.808,148.384
C00772=1203.080,347.011,-74.345,-176.143,7.811,148.384
C00773=1203.076,347.259,-74.378,-176.141,7.814,148.385
C00774=1203.073,347.507,-74.410,-176.139,7.817,148.385
C00775=1203.068,347.754,-74.443,-176.137,7.820,148.385
C00776=1203.063,348.003,-74.476,-176.136,7.823,148.385
C00777=1203.060,348.250,-74.508,-176.133,7.826,148.385
C00778=1203.056,348.498,-74.541,-176.131,7.829,148.386
C00779=1203.051,348.746,-74.574,-176.129,7.832,148.386
C00780=1203.047,348.994,-74.606,-176.127,7.835,148.386
C00781=1203.044,349.242,-74.639,-176.125,7.838,148.386
C00782=1203.039,349.490,-74.672,-176.123,7.841,148.386
C00783=1203.034,349.737,-74.704,-176.121,7.844,148.387
C00784=1203.031,349.985,-74.736,-176.119,7.848,148.387
C00785=1203.027,350.233,-74.769,-176.118,7.850,148.387
C00786=1203.022,350.481,-74.802,-176.115,7.854,148.387
C00787=1203.018,350.728,-74.835,-176.113,7.857,148.388
C00788=1203.014,350.977,-74.868,-176.112,7.860,148.388
C00789=1203.010,351.224,-74.900,-176.109,7.863,148.388
C00790=1203.006,351.472,-74.933,-176.108,7.866,148.388
C00791=1203.002,351.720,-74.966,-176.106,7.869,148.389
C00792=1202.998,351.968,-74.999,-176.104,7.872,148.389
C00793=1202.994,352.216,-75.032,-176.102,7.875,148.389
C00794=1202.990,352.464,-75.064,-176.100,7.878,148.389
C00795=1202.985,352.711,-75.097,-176.098,7.882,148.390
C00796=1202.981,352.959,-75.130,-176.096,7.884,148.390
C00797=1202.977,353.206,-75.163,-176.094,7.888,148.390
C00798=1202.972,353.455,-75.196,-176.092,7.890,148.390
C00799=1202.968,353.702,-75.229,-176.090,7.894,148.391
C00800=1202.965,353.950,-75.261,-176.089,7.897,148.391
C00801=1202.961,354.198,-75.294,-176.087,7.900,148.391
C00802=1202.957,354.445,-75.328,-176.085,7.903,148.391
C00803=1202.952,354.694,-75.360,-176.083,7.907,148.392
C00804=1202.948,354.941,-75.393,-176.081,7.909,148.392
C00805=1202.944,355.189,-75.426,-176.079,7.913,148.392
C00806=1202.940,355.437,-75.459,-176.077,7.915,148.392
C00807=1202.936,355.685,-75.493,-176.076,7.919,148.393
C00808=1202.931,355.932,-75.526,-176.073,7.922,148.393
C00809=1202.927,356.180,-75.559,-176.072,7.925,148.393
C00810=1202.924,356.427,-75.592,-176.070,7.928,148.394
C00811=1202.919,356.676,-75.624,-176.068,7.931,148.394
C00812=1202.915,356.923,-75.657,-176.066,7.934,148.394
C00813=1202.911,357.171,-75.690,-176.064,7.938,148.395
C00814=1202.907,357.419,-75.723,-176.063,7.940,148.395
C00815=1202.903,357.667,-75.757,-176.061,7.944,148.395
C00816=1202.899,357.914,-75.790,-176.059,7.946,148.395
C00817=1202.895,358.162,-75.823,-176.057,7.950,148.396
C00818=1202.891,358.410,-75.856,-176.055,7.953,148.396
C00819=1202.886,358.658,-75.889,-176.053,7.956,148.396
C00820=1202.882,358.905,-75.922,-176.052,7.960,148.397
C00821=1202.879,359.154,-75.956,-176.050,7.962,148.397
C00822=1202.875,359.401,-75.989,-176.048,7.966,148.397
C00823=1202.870,359.649,-76.022,-176.046,7.969,148.397
C00824=1202.866,359.897,-76.055,-176.045,7.972,148.398
C00825=1202.862,360.145,-76.088,-176.043,7.975,148.398
C00826=1202.858,360.392,-76.122,-176.041,7.978,148.398
C00827=1202.854,360.639,-76.156,-176.039,7.981,148.399
C00828=1202.850,360.887,-76.189,-176.038,7.984,148.399
C00829=1202.846,361.135,-76.222,-176.036,7.988,148.399
C00830=1202.841,361.383,-76.256,-176.035,7.990,148.400
C00831=1202.837,361.631,-76.289,-176.033,7.994,148.400
C00832=1202.833,361.878,-76.322,-176.031,7.997,148.400
C00833=1202.829,362.127,-76.355,-176.029,8.000,148.401
C00834=1202.825,362.374,-76.389,-176.027,8.003,148.401
C00835=1202.821,362.622,-76.422,-176.026,8.006,148.401
C00836=1202.817,362.869,-76.456,-176.024,8.010,148.402
C00837=1202.813,363.117,-76.489,-176.023,8.012,148.402
C00838=1202.809,363.365,-76.522,-176.021,8.016,148.402
C00839=1202.805,363.612,-76.556,-176.020,8.019,148.403
C00840=1202.800,363.860,-76.590,-176.017,8.022,148.403
C00841=1202.797,364.108,-76.623,-176.016,8.025,148.403
C00842=1202.792,364.356,-76.656,-176.014,8.029,148.404
C00843=1202.789,364.603,-76.690,-176.013,8.031,148.404
C00844=1202.784,364.851,-76.723,-176.011,8.035,148.405
C00845=1202.780,365.099,-76.756,-176.010,8.038,148.405
C00846=1202.776,365.346,-76.790,-176.008,8.041,148.405
C00847=1202.772,365.595,-76.824,-176.006,8.044,148.406
C00848=1202.768,365.842,-76.858,-176.005,8.047,148.406
C00849=1202.764,366.089,-76.891,-176.003,8.050,148.406
C00850=1202.759,366.371,-76.929,-176.002,8.054,148.407
C00851=1202.755,366.651,-76.967,-176.000,8.057,148.407
C00852=1202.750,366.932,-77.006,-175.998,8.061,148.408
C00853=1202.746,367.212,-77.044,-175.997,8.064,148.408
C00854=1202.742,367.460,-77.077,-175.995,8.068,148.409
C00855=1202.737,367.708,-77.110,-175.993,8.070,148.409
C00856=1202.734,367.955,-77.144,-175.992,8.074,148.409
C00857=1202.729,368.203,-77.178,-175.990,8.077,148.410
C00858=1202.726,368.451,-77.212,-175.989,8.079,148.410
C00859=1202.721,368.698,-77.245,-175.987,8.083,148.410
C00860=1202.718,368.945,-77.279,-175.986,8.086,148.411
C00861=1202.713,369.194,-77.313,-175.984,8.089,148.411
C00862=1202.709,369.441,-77.346,-175.983,8.092,148.412
C00863=1202.705,369.689,-77.380,-175.982,8.095,148.412
C00864=1202.700,369.937,-77.414,-175.980,8.099,148.412
C00865=1202.697,370.184,-77.448,-175.979,8.101,148.413
C00866=1202.692,370.432,-77.481,-175.978,8.104,148.413
C00867=1202.688,370.680,-77.516,-175.976,8.108,148.414
C00868=1202.685,370.927,-77.550,-175.975,8.111,148.414
C00869=1202.681,371.175,-77.583,-175.974,8.114,148.414
C00870=1202.676,371.422,-77.618,-175.972,8.117,148.415
C00871=1202.672,371.671,-77.651,-175.971,8.120,148.415
C00872=1202.669,371.918,-77.685,-175.969,8.123,148.416
C00873=1202.664,372.166,-77.719,-175.968,8.126,148.416
C00874=1202.660,372.413,-77.753,-175.966,8.129,148.416
C00875=1202.657,372.661,-77.787,-175.965,8.132,148.417
C00876=1202.652,372.909,-77.821,-175.964,8.135,148.417
C00877=1202.648,373.156,-77.854,-175.962,8.139,148.418
C00878=1202.643,373.404,-77.888,-175.961,8.142,148.418
C00879=1202.640,373.652,-77.922,-175.960,8.144,148.419
C00880=1202.636,373.899,-77.956,-175.959,8.147,148.419
C00881=1202.631,374.147,-77.990,-175.957,8.151,148.419
C00882=1202.628,374.395,-78.024,-175.956,8.154,148.420
C00883=1202.623,374.642,-78.059,-175.955,8.156,148.420
C00884=1202.619,374.890,-78.092,-175.954,8.160,148.421
C00885=1202.615,375.137,-78.126,-175.953,8.162,148.421
C00886=1202.611,375.385,-78.161,-175.951,8.166,148.422
C00887=1202.608,375.632,-78.194,-175.950,8.169,148.422
C00888=1202.603,375.880,-78.228,-175.949,8.172,148.422
C00889=1202.599,376.128,-78.262,-175.948,8.175,148.423
C00890=1202.595,376.376,-78.297,-175.947,8.178,148.423
C00891=1202.591,376.623,-78.330,-175.945,8.180,148.424
C00892=1202.587,376.871,-78.365,-175.944,8.184,148.424
C00893=1202.583,377.118,-78.399,-175.943,8.187,148.425
C00894=1202.578,377.366,-78.433,-175.942,8.190,148.425
C00895=1202.575,377.614,-78.467,-175.941,8.193,148.426
C00896=1202.570,377.862,-78.501,-175.940,8.196,148.426
C00897=1202.566,378.109,-78.535,-175.938,8.199,148.427
C00898=1202.562,378.357,-78.570,-175.938,8.202,148.427
C00899=1202.559,378.604,-78.604,-175.936,8.205,148.428
C00900=1202.554,378.851,-78.638,-175.935,8.207,148.428
C00901=1202.551,379.100,-78.672,-175.934,8.210,148.429
C00902=1202.546,379.347,-78.706,-175.933,8.214,148.429
C00903=1202.542,379.594,-78.740,-175.931,8.217,148.429
C00904=1202.538,379.843,-78.775,-175.931,8.220,148.430
C00905=1202.534,380.090,-78.809,-175.929,8.223,148.430
C00906=1202.530,380.338,-78.844,-175.929,8.226,148.431
C00907=1202.527,380.585,-78.878,-175.928,8.229,148.431
C00908=1202.522,380.832,-78.912,-175.927,8.232,148.432
C00909=1202.519,381.080,-78.946,-175.926,8.235,148.432
C00910=1202.514,381.328,-78.980,-175.925,8.238,148.433
C00911=1202.509,381.576,-79.014,-175.924,8.241,148.433
C00912=1202.506,381.823,-79.049,-175.923,8.244,148.434
C00913=1202.501,382.071,-79.083,-175.922,8.246,148.434
C00914=1202.498,382.319,-79.117,-175.921,8.249,148.435
C00915=1202.494,382.566,-79.152,-175.920,8.252,148.435
C00916=1202.489,382.813,-79.186,-175.919,8.255,148.436
C00917=1202.486,383.061,-79.221,-175.918,8.257,148.436
C00918=1202.481,383.309,-79.255,-175.917,8.261,148.437
C00919=1202.478,383.557,-79.289,-175.916,8.263,148.437
C00920=1202.473,383.804,-79.324,-175.915,8.266,148.438
C00921=1202.469,384.051,-79.358,-175.914,8.269,148.438
C00922=1202.466,384.299,-79.392,-175.913,8.272,148.439
C00923=1202.461,384.547,-79.427,-175.913,8.275,148.439
C00924=1202.457,384.795,-79.462,-175.912,8.277,148.440
C00925=1202.453,385.042,-79.496,-175.911,8.281,148.440
C00926=1202.449,385.290,-79.530,-175.910,8.283,148.441
C00927=1202.445,385.537,-79.565,-175.909,8.286,148.441
C00928=1202.441,385.784,-79.599,-175.908,8.290,148.442
C00929=1202.437,386.033,-79.634,-175.907,8.292,148.442
C00930=1202.433,386.279,-79.669,-175.907,8.295,148.443
C00931=1202.429,386.527,-79.703,-175.906,8.298,148.443
C00932=1202.425,386.775,-79.737,-175.905,8.301,148.444
C00933=1202.421,387.023,-79.772,-175.904,8.304,148.444
C00934=1202.417,387.270,-79.806,-175.904,8.306,148.445
C00935=1202.413,387.518,-79.841,-175.903,8.309,148.445
C00936=1202.409,387.765,-79.875,-175.902,8.312,148.446
C00937=1202.405,388.013,-79.910,-175.901,8.315,148.446
C00938=1202.401,388.261,-79.944,-175.901,8.317,148.447
C00939=1202.397,388.507,-79.979,-175.900,8.320,148.447
C00940=1202.393,388.756,-80.014,-175.899,8.323,148.448
C00941=1202.389,389.003,-80.048,-175.899,8.325,148.449
C00942=1202.385,389.251,-80.083,-175.898,8.328,148.449
C00943=1202.380,389.498,-80.117,-175.897,8.331,148.450
C00944=1202.377,389.746,-80.152,-175.897,8.334,148.450
C00945=1202.373,389.993,-80.187,-175.896,8.337,148.451
C00946=1202.369,390.241,-80.222,-175.895,8.339,148.451
C00947=1202.364,390.488,-80.256,-175.894,8.342,148.452
C00948=1202.361,390.736,-80.290,-175.894,8.345,148.452
C00949=1202.357,390.983,-80.325,-175.893,8.347,148.453
C00950=1202.353,391.231,-80.360,-175.892,8.350,148.453
C00951=1202.348,391.478,-80.395,-175.891,8.353,148.454
C00952=1202.345,391.726,-80.429,-175.891,8.355,148.454
C00953=1202.340,391.974,-80.463,-175.890,8.358,148.455
C00954=1202.336,392.256,-80.503,-175.890,8.362,148.455
C00955=1202.331,392.539,-80.544,-175.889,8.365,148.456
C00956=1202.326,392.822,-80.583,-175.889,8.367,148.457
C00957=1202.322,393.104,-80.623,-175.888,8.370,148.457
C00958=1202.318,393.352,-80.657,-175.887,8.373,148.458
C00959=1202.314,393.600,-80.692,-175.887,8.375,148.458
C00960=1202.310,393.848,-80.727,-175.886,8.378,148.459
C00961=1202.307,394.095,-80.762,-175.885,8.380,148.459
C00962=1202.302,394.342,-80.796,-175.885,8.384,148.460
C00963=1202.298,394.590,-80.831,-175.884,8.386,148.460
C00964=1202.294,394.837,-80.866,-175.884,8.389,148.461
C00965=1202.290,395.085,-80.901,-175.883,8.391,148.461
C00966=1202.285,395.333,-80.936,-175.883,8.394,148.462
C00967=1202.282,395.580,-80.970,-175.882,8.396,148.462
C00968=1202.278,395.827,-81.005,-175.882,8.399,148.463
C00969=1202.274,396.076,-81.040,-175.881,8.402,148.463
C00970=1202.270,396.322,-81.075,-175.881,8.404,148.464
C00971=1202.266,396.570,-81.110,-175.880,8.407,148.465
C00972=1202.261,396.817,-81.145,-175.880,8.409,148.465
C00973=1202.257,397.065,-81.180,-175.879,8.411,148.465
C00974=1202.254,397.313,-81.214,-175.878,8.414,148.466
C00975=1202.250,397.560,-81.249,-175.878,8.417,148.467
C00976=1202.246,397.808,-81.284,-175.878,8.419,148.467
C00977=1202.242,398.055,-81.319,-175.877,8.422,148.468
C00978=1202.238,398.303,-81.354,-175.877,8.424,148.468
C00979=1202.233,398.550,-81.389,-175.877,8.427,148.469
C00980=1202.230,398.798,-81.424,-175.875,8.429,148.469
C00981=1202.226,399.046,-81.459,-175.875,8.432,148.470
C00982=1202.222,399.293,-81.494,-175.875,8.434,148.470
C00983=1202.218,399.541,-81.528,-175.874,8.437,148.471
C00984=1202.214,399.787,-81.564,-175.874,8.439,148.471
C00985=1202.210,400.036,-81.598,-175.874,8.441,148.472
C00986=1202.205,400.283,-81.633,-175.874,8.444,148.472
C00987=1202.202,400.531,-81.668,-175.873,8.447,148.473
C00988=1202.198,400.779,-81.703,-175.872,8.449,148.473
C00989=1202.193,401.025,-81.738,-175.872,8.451,148.474
C00990=1202.189,401.274,-81.773,-175.872,8.453,148.474
C00991=1202.185,401.520,-81.808,-175.871,8.456,148.475
C00992=1202.181,401.768,-81.843,-175.871,8.459,148.476
C00993=1202.177,402.015,-81.878,-175.870,8.461,148.476
C00994=1202.173,402.263,-81.913,-175.870,8.463,148.477
C00995=1202.170,402.511,-81.948,-175.870,8.466,148.477
C00996=1202.165,402.758,-81.983,-175.869,8.468,148.477
C00997=1202.162,403.005,-82.018,-175.869,8.471,148.478
C00998=1202.157,403.253,-82.053,-175.868,8.473,148.479
C00999=1202.154,403.500,-82.088,-175.868,8.475,148.479
C01000=1202.150,403.748,-82.124,-175.868,8.477,148.480
C01001=1202.145,403.995,-82.158,-175.867,8.481,148.480
C01002=1202.142,404.243,-82.194,-175.867,8.483,148.481
C01003=1202.138,404.491,-82.229,-175.867,8.485,148.481
C01004=1202.133,404.738,-82.264,-175.866,8.487,148.482
C01005=1202.129,404.986,-82.299,-175.866,8.489,148.482
C01006=1202.125,405.233,-82.334,-175.866,8.492,148.483
C01007=1202.121,405.481,-82.369,-175.865,8.494,148.483
C01008=1202.118,405.728,-82.404,-175.865,8.496,148.484
C01009=1202.113,405.975,-82.439,-175.865,8.498,148.484
C01010=1202.109,406.223,-82.474,-175.864,8.501,148.485
C01011=1202.106,406.471,-82.510,-175.863,8.503,148.485
C01012=1202.101,406.718,-82.544,-175.863,8.506,148.486
C01013=1202.097,406.966,-82.580,-175.863,8.508,148.486
C01014=1202.093,407.212,-82.615,-175.863,8.510,148.487
C01015=1202.089,407.461,-82.650,-175.862,8.513,148.487
C01016=1202.086,407.708,-82.685,-175.862,8.515,148.488
C01017=1202.081,407.955,-82.721,-175.862,8.517,148.488
C01018=1202.077,408.203,-82.755,-175.861,8.519,148.489
C01019=1202.074,408.450,-82.791,-175.861,8.521,148.489
C01020=1202.069,408.698,-82.825,-175.861,8.524,148.490
C01021=1202.065,408.945,-82.861,-175.861,8.526,148.490
C01022=1202.062,409.193,-82.896,-175.860,8.528,148.491
C01023=1202.057,409.440,-82.931,-175.860,8.530,148.491
C01024=1202.053,409.688,-82.966,-175.860,8.532,148.492
C01025=1202.050,409.935,-83.002,-175.859,8.535,148.492
C01026=1202.045,410.183,-83.036,-175.859,8.537,148.493
C01027=1202.042,410.430,-83.072,-175.859,8.539,148.493
C01028=1202.038,410.678,-83.108,-175.859,8.541,148.494
C01029=1202.033,410.925,-83.142,-175.858,8.544,148.494
C01030=1202.030,411.173,-83.178,-175.858,8.546,148.495
C01031=1202.026,411.420,-83.213,-175.858,8.548,148.495
C01032=1202.021,411.667,-83.249,-175.857,8.550,148.496
C01033=1202.017,411.915,-83.284,-175.857,8.552,148.496
C01034=1202.013,412.163,-83.319,-175.857,8.555,148.497
C01035=1202.009,412.410,-83.354,-175.856,8.557,148.497
C01036=1202.005,412.658,-83.389,-175.856,8.559,148.498
C01037=1202.002,412.905,-83.425,-175.856,8.561,148.498
C01038=1201.997,413.152,-83.460,-175.855,8.563,148.499
C01039=1201.994,413.400,-83.496,-175.856,8.565,148.499
C01040=1201.990,413.648,-83.530,-175.855,8.567,148.500
C01041=1201.985,413.895,-83.566,-175.855,8.569,148.500
C01042=1201.982,414.142,-83.601,-175.855,8.571,148.501
C01043=1201.978,414.390,-83.637,-175.854,8.574,148.501
C01044=1201.973,414.637,-83.672,-175.854,8.576,148.502
C01045=1201.969,414.885,-83.707,-175.854,8.578,148.502
C01046=1201.965,415.132,-83.743,-175.853,8.580,148.502
C01047=1201.962,415.380,-83.778,-175.853,8.582,148.503
C01048=1201.957,415.627,-83.814,-175.853,8.584,148.503
C01049=1201.953,415.875,-83.848,-175.853,8.586,148.504
C01050=1201.948,416.181,-83.893,-175.852,8.589,148.504
C01051=1201.945,416.487,-83.936,-175.852,8.592,148.505
C01052=1201.943,416.794,-83.980,-175.852,8.594,148.506
C01053=1201.946,417.099,-84.023,-175.852,8.596,148.506
C01054=1201.524,417.100,-84.061,-175.855,8.607,148.510
C01055=1201.522,416.791,-84.018,-175.855,8.604,148.509
C01056=1201.522,416.482,-83.974,-175.855,8.602,148.509
C01057=1201.527,416.172,-83.930,-175.855,8.600,148.508
C01058=1201.532,415.863,-83.885,-175.856,8.596,148.508
C01059=1201.536,415.616,-83.850,-175.856,8.594,148.507
C01060=1201.540,415.369,-83.815,-175.856,8.593,148.507
C01061=1201.544,415.122,-83.779,-175.857,8.591,148.506
C01062=1201.547,414.874,-83.744,-175.857,8.589,148.506
C01063=1201.553,414.626,-83.709,-175.857,8.586,148.505
C01064=1201.556,414.379,-83.673,-175.858,8.584,148.505
C01065=1201.560,414.131,-83.638,-175.858,8.582,148.504
C01066=1201.564,413.884,-83.602,-175.858,8.580,148.504
C01067=1201.568,413.636,-83.567,-175.858,8.578,148.503
C01068=1201.572,413.389,-83.532,-175.859,8.575,148.503
C01069=1201.575,413.141,-83.496,-175.859,8.574,148.502
C01070=1201.580,412.895,-83.461,-175.859,8.572,148.502
C01071=1201.584,412.646,-83.426,-175.859,8.570,148.501
C01072=1201.587,412.399,-83.391,-175.859,8.567,148.501
C01073=1201.592,412.152,-83.356,-175.860,8.565,148.500
C01074=1201.595,411.905,-83.320,-175.860,8.563,148.500
C01075=1201.600,411.656,-83.285,-175.861,8.561,148.499
C01076=1201.604,411.409,-83.249,-175.861,8.559,148.499
C01077=1201.608,411.162,-83.214,-175.861,8.556,148.498
C01078=1201.612,410.914,-83.179,-175.861,8.554,148.498
C01079=1201.616,410.667,-83.144,-175.861,8.552,148.497
C01080=1201.620,410.419,-83.108,-175.862,8.550,148.497
C01081=1201.623,410.172,-83.073,-175.862,8.548,148.496
C01082=1201.628,409.925,-83.038,-175.863,8.545,148.496
C01083=1201.632,409.677,-83.003,-175.863,8.543,148.495
C01084=1201.635,409.430,-82.967,-175.863,8.541,148.495
C01085=1201.640,409.182,-82.933,-175.863,8.538,148.494
C01086=1201.644,408.935,-82.897,-175.864,8.536,148.494
C01087=1201.647,408.687,-82.862,-175.864,8.534,148.493
C01088=1201.652,408.440,-82.827,-175.864,8.532,148.493
C01089=1201.656,408.192,-82.792,-175.865,8.530,148.492
C01090=1201.659,407.945,-82.756,-175.865,8.527,148.492
C01091=1201.664,407.697,-82.722,-175.865,8.525,148.491
C01092=1201.667,407.450,-82.686,-175.865,8.523,148.491
C01093=1201.671,407.202,-82.651,-175.866,8.521,148.490
C01094=1201.676,406.955,-82.616,-175.866,8.519,148.490
C01095=1201.679,406.707,-82.581,-175.866,8.516,148.489
C01096=1201.684,406.460,-82.546,-175.867,8.514,148.489
C01097=1201.688,406.212,-82.511,-175.867,8.512,148.488
C01098=1201.692,405.964,-82.476,-175.867,8.510,148.488
C01099=1201.696,405.718,-82.441,-175.867,8.507,148.487
C01100=1201.699,405.470,-82.405,-175.868,8.504,148.487
C01101=1201.703,405.222,-82.370,-175.869,8.502,148.486
C01102=1201.708,404.975,-82.335,-175.869,8.500,148.486
C01103=1201.712,404.727,-82.300,-175.869,8.498,148.485
C01104=1201.716,404.480,-82.265,-175.869,8.495,148.485
C01105=1201.720,404.233,-82.229,-175.870,8.493,148.484
C01106=1201.724,403.985,-82.195,-175.870,8.491,148.484
C01107=1201.728,403.738,-82.159,-175.870,8.489,148.483
C01108=1201.732,403.490,-82.125,-175.871,8.486,148.483
C01109=1201.735,403.242,-82.089,-175.872,8.484,148.482
C01110=1201.740,402.995,-82.055,-175.872,8.481,148.482
C01111=1201.744,402.747,-82.019,-175.872,8.479,148.481
C01112=1201.748,402.500,-81.985,-175.872,8.477,148.481
C01113=1201.752,402.252,-81.949,-175.872,8.474,148.480
C01114=1201.756,402.004,-81.914,-175.873,8.471,148.480
C01115=1201.760,401.757,-81.879,-175.873,8.469,148.479
C01116=1201.764,401.509,-81.844,-175.874,8.467,148.478
C01117=1201.768,401.262,-81.809,-175.874,8.465,148.478
C01118=1201.772,401.014,-81.774,-175.875,8.462,148.478
C01119=1201.775,400.767,-81.739,-175.875,8.459,148.477
C01120=1201.780,400.520,-81.705,-175.876,8.457,148.476
C01121=1201.783,400.272,-81.669,-175.876,8.455,148.476
C01122=1201.788,400.025,-81.635,-175.877,8.452,148.475
C01123=1201.792,399.777,-81.599,-175.877,8.450,148.475
C01124=1201.796,399.529,-81.564,-175.877,8.447,148.474
C01125=1201.800,399.282,-81.529,-175.877,8.445,148.474
C01126=1201.804,399.034,-81.494,-175.878,8.442,148.473
C01127=1201.808,398.788,-81.459,-175.879,8.440,148.473
C01128=1201.812,398.539,-81.424,-175.879,8.438,148.472
C01129=1201.816,398.293,-81.389,-175.880,8.435,148.472
C01130=1201.820,398.045,-81.355,-175.880,8.432,148.471
C01131=1201.824,397.797,-81.320,-175.880,8.430,148.471
C01132=1201.828,397.550,-81.285,-175.881,8.427,148.470
C01133=1201.832,397.302,-81.250,-175.881,8.425,148.470
C01134=1201.836,397.055,-81.215,-175.882,8.423,148.469
C01135=1201.840,396.807,-81.180,-175.883,8.420,148.469
C01136=1201.845,396.559,-81.146,-175.883,8.417,148.468
C01137=1201.848,396.312,-81.110,-175.883,8.415,148.468
C01138=1201.852,396.065,-81.076,-175.884,8.412,148.467
C01139=1201.856,395.817,-81.041,-175.884,8.410,148.466
C01140=1201.860,395.570,-81.006,-175.885,8.407,148.466
C01141=1201.864,395.322,-80.971,-175.885,8.405,148.466
C01142=1201.868,395.074,-80.936,-175.886,8.402,148.465
C01143=1201.873,394.827,-80.901,-175.886,8.399,148.464
C01144=1201.876,394.579,-80.867,-175.887,8.397,148.464
C01145=1201.880,394.332,-80.832,-175.887,8.394,148.463
C01146=1201.884,394.084,-80.797,-175.888,8.392,148.463
C01147=1201.889,393.837,-80.763,-175.888,8.389,148.462
C01148=1201.893,393.589,-80.728,-175.889,8.387,148.462
C01149=1201.897,393.342,-80.693,-175.890,8.383,148.461
C01150=1201.900,393.094,-80.658,-175.890,8.381,148.461
C01151=1201.905,392.811,-80.618,-175.891,8.378,148.460
C01152=1201.910,392.528,-80.579,-175.892,8.375,148.459
C01153=1201.914,392.246,-80.539,-175.892,8.372,148.459
C01154=1201.919,391.963,-80.500,-175.893,8.369,148.458
C01155=1201.922,391.715,-80.464,-175.893,8.366,148.458
C01156=1201.927,391.468,-80.430,-175.894,8.363,148.457
C01157=1201.931,391.220,-80.395,-175.895,8.360,148.457
C01158=1201.935,390.973,-80.361,-175.896,8.358,148.456
C01159=1201.939,390.725,-80.326,-175.896,8.355,148.456
C01160=1201.943,390.478,-80.291,-175.897,8.353,148.455
C01161=1201.947,390.230,-80.256,-175.897,8.350,148.455
C01162=1201.951,389.982,-80.222,-175.898,8.347,148.454
C01163=1201.955,389.735,-80.188,-175.899,8.345,148.454
C01164=1201.959,389.488,-80.152,-175.900,8.342,148.453
C01165=1201.963,389.240,-80.118,-175.900,8.339,148.452
C01166=1201.967,388.993,-80.084,-175.901,8.336,148.452
C01167=1201.971,388.744,-80.049,-175.902,8.333,148.452
C01168=1201.975,388.497,-80.014,-175.903,8.330,148.451
C01169=1201.980,388.250,-79.980,-175.903,8.328,148.450
C01170=1201.983,388.002,-79.945,-175.904,8.325,148.450
C01171=1201.987,387.755,-79.911,-175.905,8.322,148.449
C01172=1201.991,387.507,-79.876,-175.906,8.319,148.449
C01173=1201.995,387.260,-79.842,-175.906,8.317,148.448
C01174=1201.999,387.012,-79.807,-175.907,8.314,148.448
C01175=1202.004,386.764,-79.773,-175.908,8.311,148.447
C01176=1202.008,386.516,-79.738,-175.909,8.308,148.447
C01177=1202.011,386.269,-79.704,-175.909,8.306,148.446
C01178=1202.015,386.021,-79.668,-175.910,8.303,148.446
C01179=1202.020,385.774,-79.634,-175.911,8.300,148.445
C01180=1202.023,385.527,-79.600,-175.912,8.297,148.445
C01181=1202.027,385.279,-79.565,-175.913,8.294,148.444
C01182=1202.032,385.031,-79.531,-175.913,8.291,148.444
C01183=1202.035,384.784,-79.496,-175.914,8.289,148.443
C01184=1202.040,384.536,-79.462,-175.915,8.286,148.443
C01185=1202.044,384.288,-79.427,-175.916,8.283,148.442
C01186=1202.048,384.041,-79.393,-175.917,8.280,148.442
C01187=1202.052,383.794,-79.359,-175.918,8.277,148.441
C01188=1202.055,383.546,-79.325,-175.919,8.274,148.441
C01189=1202.060,383.298,-79.290,-175.919,8.271,148.440
C01190=1202.064,383.050,-79.255,-175.920,8.269,148.440
C01191=1202.068,382.803,-79.221,-175.921,8.266,148.439
C01192=1202.072,382.555,-79.187,-175.922,8.263,148.439
C01193=1202.076,382.308,-79.152,-175.923,8.260,148.438
C01194=1202.080,382.060,-79.118,-175.924,8.257,148.438
C01195=1202.084,381.812,-79.083,-175.925,8.254,148.437
C01196=1202.088,381.565,-79.049,-175.926,8.251,148.437
C01197=1202.092,381.317,-79.015,-175.927,8.248,148.436
C01198=1202.096,381.070,-78.981,-175.928,8.245,148.436
C01199=1202.100,380.823,-78.946,-175.929,8.242,148.435
C01200=1202.104,380.574,-78.911,-175.930,8.239,148.435
C01201=1202.108,380.327,-78.878,-175.931,8.236,148.434
C01202=1202.113,380.079,-78.844,-175.932,8.233,148.434
C01203=1202.116,379.831,-78.810,-175.933,8.230,148.433
C01204=1202.121,379.584,-78.775,-175.934,8.227,148.433
C01205=1202.124,379.336,-78.741,-175.935,8.224,148.432
C01206=1202.129,379.089,-78.706,-175.936,8.221,148.432
C01207=1202.132,378.842,-78.673,-175.938,8.219,148.432
C01208=1202.136,378.594,-78.638,-175.938,8.215,148.431
C01209=1202.141,378.346,-78.604,-175.940,8.212,148.431
C01210=1202.145,378.098,-78.570,-175.941,8.209,148.430
C01211=1202.149,377.850,-78.535,-175.942,8.206,148.430
C01212=1202.153,377.603,-78.501,-175.943,8.203,148.429
C01213=1202.157,377.356,-78.467,-175.944,8.200,148.429
C01214=1202.161,377.107,-78.433,-175.945,8.197,148.428
C01215=1202.166,376.860,-78.399,-175.947,8.194,148.428
C01216=1202.169,376.613,-78.365,-175.948,8.192,148.427
C01217=1202.173,376.365,-78.331,-175.949,8.188,148.427
C01218=1202.178,376.117,-78.297,-175.950,8.185,148.426
C01219=1202.181,375.870,-78.263,-175.951,8.182,148.426
C01220=1202.185,375.622,-78.228,-175.952,8.179,148.425
C01221=1202.189,375.375,-78.195,-175.953,8.176,148.425
C01222=1202.194,375.127,-78.161,-175.955,8.173,148.425
C01223=1202.197,374.879,-78.127,-175.956,8.170,148.424
C01224=1202.202,374.631,-78.092,-175.958,8.167,148.424
C01225=1202.206,374.384,-78.058,-175.958,8.164,148.423
C01226=1202.210,374.137,-78.025,-175.960,8.161,148.423
C01227=1202.214,373.888,-77.990,-175.961,8.157,148.422
C01228=1202.218,373.641,-77.956,-175.963,8.155,148.422
C01229=1202.222,373.393,-77.923,-175.964,8.152,148.422
C01230=1202.226,373.145,-77.888,-175.965,8.149,148.421
C01231=1202.230,372.898,-77.855,-175.966,8.145,148.421
C01232=1202.234,372.650,-77.821,-175.968,8.142,148.420
C01233=1202.238,372.403,-77.787,-175.969,8.139,148.420
C01234=1202.243,372.154,-77.753,-175.970,8.137,148.419
C01235=1202.246,371.907,-77.719,-175.972,8.133,148.419
C01236=1202.250,371.660,-77.686,-175.973,8.130,148.419
C01237=1202.255,371.412,-77.651,-175.974,8.127,148.418
C01238=1202.258,371.164,-77.617,-175.976,8.124,148.418
C01239=1202.262,370.917,-77.584,-175.977,8.121,148.417
C01240=1202.267,370.669,-77.549,-175.978,8.118,148.417
C01241=1202.271,370.421,-77.516,-175.980,8.114,148.417
C01242=1202.274,370.174,-77.482,-175.981,8.112,148.416
C01243=1202.279,369.926,-77.448,-175.983,8.109,148.416
C01244=1202.283,369.679,-77.414,-175.984,8.105,148.415
C01245=1202.287,369.431,-77.381,-175.986,8.102,148.415
C01246=1202.291,369.183,-77.346,-175.987,8.100,148.415
C01247=1202.295,368.935,-77.313,-175.989,8.096,148.414
C01248=1202.299,368.688,-77.279,-175.990,8.093,148.414
C01249=1202.303,368.440,-77.246,-175.992,8.089,148.413
C01250=1202.308,368.193,-77.212,-175.993,8.087,148.413
C01251=1202.311,367.944,-77.178,-175.994,8.084,148.412
C01252=1202.316,367.697,-77.145,-175.996,8.080,148.412
C01253=1202.319,367.449,-77.111,-175.997,8.078,148.412
C01254=1202.324,367.201,-77.077,-175.999,8.074,148.411
C01255=1202.328,366.921,-77.040,-176.000,8.071,148.411
C01256=1202.333,366.640,-77.001,-176.002,8.068,148.411
C01257=1202.338,366.360,-76.963,-176.004,8.064,148.410
C01258=1202.342,366.079,-76.925,-176.006,8.060,148.410
C01259=1202.347,365.832,-76.891,-176.008,8.057,148.409
C01260=1202.351,365.584,-76.858,-176.009,8.054,148.409
C01261=1202.354,365.335,-76.824,-176.011,8.051,148.409
C01262=1202.358,365.088,-76.790,-176.012,8.048,148.408
C01263=1202.362,364.841,-76.757,-176.014,8.044,148.408
C01264=1202.366,364.593,-76.724,-176.015,8.041,148.407
C01265=1202.371,364.345,-76.690,-176.017,8.039,148.407
C01266=1202.375,364.098,-76.656,-176.019,8.035,148.407
C01267=1202.379,363.850,-76.623,-176.020,8.032,148.406
C01268=1202.383,363.601,-76.590,-176.022,8.029,148.406
C01269=1202.387,363.354,-76.556,-176.024,8.025,148.406
C01270=1202.391,363.107,-76.523,-176.025,8.023,148.405
C01271=1202.395,362.859,-76.490,-176.027,8.019,148.405
C01272=1202.400,362.611,-76.456,-176.028,8.016,148.405
C01273=1202.404,362.363,-76.423,-176.030,8.013,148.404
C01274=1202.408,362.116,-76.389,-176.032,8.010,148.404
C01275=1202.412,361.868,-76.356,-176.034,8.007,148.404
C01276=1202.415,361.620,-76.322,-176.035,8.004,148.403
C01277=1202.420,361.372,-76.289,-176.037,8.000,148.403
C01278=1202.424,361.124,-76.256,-176.038,7.998,148.403
C01279=1202.428,360.877,-76.223,-176.041,7.994,148.402
C01280=1202.432,360.629,-76.189,-176.042,7.991,148.402
C01281=1202.436,360.382,-76.156,-176.044,7.988,148.402
C01282=1202.440,360.134,-76.122,-176.046,7.984,148.401
C01283=1202.444,359.886,-76.089,-176.047,7.982,148.401
C01284=1202.448,359.639,-76.056,-176.049,7.978,148.401
C01285=1202.452,359.391,-76.023,-176.051,7.976,148.401
C01286=1202.456,359.143,-75.990,-176.053,7.972,148.400
C01287=1202.460,358.895,-75.956,-176.055,7.969,148.400
C01288=1202.464,358.647,-75.923,-176.056,7.966,148.400
C01289=1202.468,358.399,-75.890,-176.058,7.963,148.399
C01290=1202.472,358.152,-75.857,-176.059,7.960,148.399
C01291=1202.477,357.904,-75.824,-176.062,7.957,148.399
C01292=1202.481,357.656,-75.791,-176.064,7.953,148.398
C01293=1202.485,357.408,-75.757,-176.065,7.950,148.398
C01294=1202.489,357.161,-75.724,-176.067,7.947,148.398
C01295=1202.493,356.913,-75.691,-176.069,7.944,148.397
C01296=1202.497,356.665,-75.658,-176.071,7.941,148.397
C01297=1202.501,356.417,-75.625,-176.073,7.938,148.397
C01298=1202.506,356.170,-75.592,-176.074,7.935,148.397
C01299=1202.510,355.922,-75.558,-176.076,7.931,148.396
C01300=1202.514,355.674,-75.526,-176.078,7.929,148.396
C01301=1202.518,355.426,-75.493,-176.080,7.925,148.396
C01302=1202.522,355.178,-75.460,-176.082,7.922,148.396
C01303=1202.527,354.930,-75.427,-176.084,7.919,148.395
C01304=1202.531,354.683,-75.393,-176.085,7.916,148.395
C01305=1202.535,354.435,-75.360,-176.088,7.912,148.395
C01306=1202.538,354.188,-75.328,-176.089,7.910,148.395
C01307=1202.543,353.939,-75.295,-176.092,7.907,148.394
C01308=1202.547,353.692,-75.262,-176.093,7.904,148.394
C01309=1202.551,353.444,-75.229,-176.095,7.900,148.394
C01310=1202.555,353.196,-75.196,-176.097,7.897,148.393
C01311=1202.559,352.948,-75.163,-176.099,7.895,148.393
C01312=1202.564,352.700,-75.130,-176.101,7.891,148.393
C01313=1202.567,352.453,-75.098,-176.103,7.888,148.393
C01314=1202.571,352.205,-75.064,-176.105,7.885,148.392
C01315=1202.576,351.957,-75.032,-176.107,7.882,148.392
C01316=1202.580,351.709,-74.999,-176.109,7.878,148.392
C01317=1202.584,351.462,-74.966,-176.110,7.876,148.392
C01318=1202.588,351.214,-74.933,-176.112,7.872,148.391
C01319=1202.592,350.966,-74.901,-176.114,7.870,148.391
C01320=1202.596,350.718,-74.868,-176.116,7.866,148.391
C01321=1202.601,350.471,-74.835,-176.119,7.863,148.391
C01322=1202.605,350.222,-74.802,-176.120,7.861,148.391
C01323=1202.608,349.975,-74.770,-176.122,7.857,148.390
C01324=1202.613,349.726,-74.737,-176.124,7.854,148.390
C01325=1202.617,349.479,-74.704,-176.126,7.851,148.390
C01326=1202.622,349.232,-74.671,-176.128,7.848,148.389
C01327=1202.625,348.984,-74.640,-176.130,7.844,148.389
C01328=1202.630,348.736,-74.606,-176.132,7.842,148.389
C01329=1202.634,348.488,-74.574,-176.134,7.839,148.389
C01330=1202.637,348.240,-74.541,-176.136,7.835,148.389
C01331=1202.642,347.992,-74.509,-176.138,7.833,148.388
C01332=1202.646,347.744,-74.476,-176.140,7.829,148.388
C01333=1202.650,347.496,-74.443,-176.142,7.827,148.388
C01334=1202.654,347.249,-74.411,-176.144,7.824,148.388
C01335=1202.659,347.001,-74.379,-176.146,7.820,148.388
C01336=1202.663,346.753,-74.346,-176.148,7.818,148.387
C01337=1202.667,346.505,-74.314,-176.150,7.814,148.387
C01338=1202.671,346.257,-74.281,-176.152,7.811,148.387
C01339=1202.675,346.009,-74.248,-176.154,7.809,148.387
C01340=1202.679,345.762,-74.216,-176.156,7.805,148.387
C01341=1202.684,345.514,-74.183,-176.159,7.802,148.386
C01342=1202.688,345.266,-74.152,-176.160,7.799,148.386
C01343=1202.692,345.018,-74.118,-176.162,7.796,148.386
C01344=1202.696,344.770,-74.086,-176.165,7.793,148.386
C01345=1202.700,344.523,-74.054,-176.166,7.790,148.386
C01346=1202.705,344.275,-74.021,-176.169,7.787,148.385
C01347=1202.708,344.026,-73.990,-176.171,7.783,148.385
C01348=1202.712,343.779,-73.956,-176.172,7.781,148.385
C01349=1202.717,343.530,-73.924,-176.175,7.778,148.385
C01350=1202.721,343.283,-73.892,-176.177,7.774,148.384
C01351=1202.725,343.035,-73.859,-176.179,7.772,148.384
C01352=1202.729,342.787,-73.827,-176.181,7.768,148.384
C01353=1202.733,342.539,-73.795,-176.183,7.765,148.384
C01354=1202.738,342.292,-73.764,-176.185,7.763,148.384
C01355=1202.742,342.044,-73.730,-176.187,7.760,148.384
C01356=1202.746,341.796,-73.699,-176.190,7.756,148.383
C01357=1202.750,341.547,-73.666,-176.191,7.754,148.383
C01358=1202.755,341.300,-73.634,-176.193,7.750,148.383
C01359=1202.759,341.022,-73.598,-176.196,7.747,148.383
C01360=1202.763,340.743,-73.561,-176.198,7.744,148.383
C01361=1202.768,340.465,-73.525,-176.200,7.740,148.382
C01362=1202.773,340.186,-73.489,-176.203,7.737,148.382
C01363=1202.777,339.939,-73.458,-176.205,7.734,148.382
C01364=1202.782,339.691,-73.425,-176.207,7.731,148.382
C01365=1202.785,339.443,-73.393,-176.209,7.728,148.382
C01366=1202.790,339.195,-73.361,-176.211,7.725,148.382
C01367=1202.794,338.947,-73.329,-176.214,7.722,148.382
C01368=1202.798,338.699,-73.297,-176.215,7.719,148.381
C01369=1202.802,338.451,-73.265,-176.218,7.716,148.381
C01370=1202.806,338.204,-73.233,-176.220,7.713,148.381
C01371=1202.811,337.955,-73.201,-176.222,7.710,148.381
C01372=1202.815,337.707,-73.169,-176.224,7.707,148.381
C01373=1202.819,337.460,-73.137,-176.226,7.704,148.381
C01374=1202.823,337.211,-73.105,-176.228,7.701,148.380
C01375=1202.827,336.963,-73.073,-176.231,7.698,148.380
C01376=1202.831,336.716,-73.042,-176.233,7.695,148.380
C01377=1202.836,336.468,-73.009,-176.235,7.691,148.380
C01378=1202.839,336.220,-72.977,-176.237,7.689,148.380
C01379=1202.844,335.972,-72.946,-176.240,7.686,148.380
C01380=1202.848,335.724,-72.914,-176.242,7.683,148.380
C01381=1202.852,335.476,-72.882,-176.244,7.680,148.379
C01382=1202.856,335.229,-72.850,-176.246,7.677,148.379
C01383=1202.861,334.980,-72.818,-176.248,7.674,148.379
C01384=1202.864,334.732,-72.786,-176.250,7.671,148.379
C01385=1202.869,334.485,-72.754,-176.253,7.668,148.379
C01386=1202.873,334.237,-72.722,-176.255,7.665,148.379
C01387=1202.878,333.989,-72.691,-176.257,7.662,148.379
C01388=1202.881,333.741,-72.659,-176.259,7.659,148.379
C01389=1202.885,333.492,-72.628,-176.262,7.656,148.378
C01390=1202.890,333.245,-72.595,-176.263,7.653,148.378
C01391=1202.894,332.997,-72.564,-176.266,7.650,148.378
C01392=1202.898,332.749,-72.532,-176.268,7.647,148.378
C01393=1202.902,332.501,-72.501,-176.270,7.645,148.378
C01394=1202.907,332.252,-72.469,-176.272,7.642,148.378
C01395=1202.911,332.005,-72.437,-176.275,7.638,148.378
C01396=1202.915,331.757,-72.405,-176.277,7.636,148.378
C01397=1202.919,331.509,-72.374,-176.279,7.633,148.377
C01398=1202.923,331.261,-72.343,-176.282,7.630,148.377
C01399=1202.928,331.013,-72.311,-176.283,7.627,148.377
C01400=1202.932,330.765,-72.279,-176.286,7.624,148.377
C01401=1202.936,330.517,-72.248,-176.288,7.621,148.377
C01402=1202.940,330.269,-72.216,-176.290,7.618,148.377
C01403=1202.944,330.021,-72.184,-176.293,7.615,148.377
C01404=1202.948,329.773,-72.153,-176.295,7.612,148.377
C01405=1202.952,329.525,-72.122,-176.297,7.610,148.377
C01406=1202.957,329.278,-72.090,-176.299,7.606,148.376
C01407=1202.961,329.029,-72.058,-176.302,7.603,148.376
C01408=1202.965,328.782,-72.027,-176.304,7.601,148.376
C01409=1202.969,328.533,-71.996,-176.306,7.597,148.376
C01410=1202.974,328.286,-71.964,-176.308,7.594,148.376
C01411=1202.978,328.038,-71.933,-176.310,7.592,148.376
C01412=1202.982,327.790,-71.902,-176.313,7.589,148.376
C01413=1202.986,327.542,-71.870,-176.315,7.586,148.376
C01414=1202.990,327.294,-71.839,-176.317,7.583,148.376
C01415=1202.994,327.046,-71.807,-176.319,7.580,148.375
C01416=1202.999,326.798,-71.777,-176.322,7.577,148.375
C01417=1203.002,326.550,-71.745,-176.324,7.575,148.375
C01418=1203.008,326.301,-71.713,-176.326,7.571,148.375
C01419=1203.012,326.053,-71.681,-176.329,7.568,148.375
C01420=1203.016,325.805,-71.651,-176.331,7.566,148.375
C01421=1203.020,325.557,-71.619,-176.333,7.563,148.375
C01422=1203.024,325.309,-71.588,-176.336,7.560,148.375
C01423=1203.029,325.061,-71.557,-176.338,7.557,148.375
C01424=1203.032,324.814,-71.526,-176.340,7.554,148.375
C01425=1203.037,324.566,-71.495,-176.343,7.551,148.375
C01426=1203.040,324.318,-71.463,-176.344,7.549,148.375
C01427=1203.045,324.070,-71.433,-176.347,7.545,148.375
C01428=1203.049,323.821,-71.402,-176.350,7.542,148.375
C01429=1203.053,323.574,-71.370,-176.352,7.539,148.374
C01430=1203.057,323.325,-71.339,-176.354,7.537,148.374
C01431=1203.062,323.077,-71.308,-176.356,7.534,148.374
C01432=1203.066,322.830,-71.277,-176.359,7.531,148.374
C01433=1203.070,322.581,-71.246,-176.361,7.528,148.374
C01434=1203.075,322.333,-71.215,-176.363,7.525,148.374
C01435=1203.079,322.085,-71.183,-176.366,7.522,148.374
C01436=1203.083,321.837,-71.152,-176.368,7.519,148.374
C01437=1203.087,321.590,-71.122,-176.370,7.516,148.374
C01438=1203.091,321.341,-71.091,-176.373,7.513,148.374
C01439=1203.095,321.094,-71.059,-176.375,7.511,148.374
C01440=1203.100,320.846,-71.029,-176.377,7.508,148.374
C01441=1203.104,320.597,-70.998,-176.379,7.506,148.374
C01442=1203.109,320.349,-70.967,-176.382,7.502,148.374
C01443=1203.113,320.100,-70.936,-176.384,7.499,148.374
C01444=1203.116,319.853,-70.905,-176.387,7.497,148.374
C01445=1203.121,319.605,-70.874,-176.389,7.494,148.373
C01446=1203.125,319.357,-70.843,-176.391,7.491,148.373
C01447=1203.129,319.109,-70.812,-176.394,7.489,148.373
C01448=1203.134,318.861,-70.781,-176.396,7.485,148.373
C01449=1203.137,318.612,-70.751,-176.398,7.482,148.373
C01450=1203.142,318.364,-70.720,-176.401,7.480,148.373
C01451=1203.147,318.117,-70.689,-176.403,7.477,148.373
C01452=1203.151,317.868,-70.658,-176.405,7.474,148.373
C01453=1203.154,317.620,-70.628,-176.408,7.471,148.373
C01454=1203.159,317.373,-70.597,-176.410,7.468,148.373
C01455=1203.163,317.124,-70.565,-176.413,7.465,148.373
C01456=1203.167,316.876,-70.535,-176.415,7.463,148.373
C01457=1203.171,316.629,-70.504,-176.417,7.460,148.373
C01458=1203.176,316.381,-70.474,-176.420,7.456,148.373
C01459=1203.180,316.132,-70.443,-176.422,7.454,148.373
C01460=1203.184,315.884,-70.412,-176.424,7.451,148.373
C01461=1203.189,315.636,-70.382,-176.427,7.448,148.373
C01462=1203.193,315.388,-70.352,-176.429,7.446,148.373
C01463=1203.197,315.111,-70.317,-176.431,7.443,148.373
C01464=1203.202,314.836,-70.283,-176.434,7.440,148.373
C01465=1203.207,314.559,-70.249,-176.437,7.436,148.373
C01466=1203.212,314.283,-70.215,-176.440,7.433,148.373
C01467=1203.215,314.035,-70.184,-176.442,7.431,148.373
C01468=1203.220,313.787,-70.154,-176.444,7.427,148.373
C01469=1203.225,313.538,-70.123,-176.447,7.424,148.373
C01470=1203.229,313.291,-70.093,-176.449,7.422,148.373
C01471=1203.233,313.042,-70.062,-176.452,7.419,148.373
C01472=1203.237,312.794,-70.031,-176.454,7.417,148.373
C01473=1203.241,312.547,-70.001,-176.456,7.413,148.372
C01474=1203.246,312.299,-69.970,-176.459,7.410,148.372
C01475=1203.250,312.050,-69.941,-176.461,7.408,148.372
C01476=1203.254,311.802,-69.910,-176.464,7.405,148.372
C01477=1203.258,311.554,-69.880,-176.466,7.402,148.372
C01478=1203.263,311.306,-69.849,-176.468,7.400,148.372
C01479=1203.267,311.057,-69.819,-176.471,7.397,148.372
C01480=1203.271,310.810,-69.789,-176.473,7.394,148.372
C01481=1203.275,310.561,-69.758,-176.476,7.391,148.372
C01482=1203.280,310.313,-69.728,-176.478,7.388,148.372
C01483=1203.284,310.065,-69.697,-176.480,7.386,148.372
C01484=1203.288,309.817,-69.667,-176.483,7.383,148.372
C01485=1203.293,309.569,-69.637,-176.485,7.380,148.372
C01486=1203.297,309.321,-69.607,-176.487,7.378,148.372
C01487=1203.301,309.073,-69.576,-176.490,7.375,148.372
C01488=1203.305,308.824,-69.546,-176.493,7.372,148.372
C01489=1203.310,308.576,-69.516,-176.495,7.369,148.372
C01490=1203.314,308.328,-69.486,-176.498,7.366,148.372
C01491=1203.318,308.080,-69.455,-176.500,7.363,148.372
C01492=1203.322,307.832,-69.425,-176.502,7.361,148.372
C01493=1203.327,307.584,-69.396,-176.505,7.358,148.372
C01494=1203.331,307.336,-69.365,-176.507,7.356,148.372
C01495=1203.335,307.088,-69.336,-176.509,7.353,148.372
C01496=1203.339,306.839,-69.304,-176.512,7.350,148.372
C01497=1203.343,306.591,-69.275,-176.514,7.347,148.372
C01498=1203.348,306.343,-69.244,-176.517,7.344,148.372
C01499=1203.352,306.095,-69.215,-176.520,7.341,148.372
C01500=1203.356,305.847,-69.185,-176.522,7.339,148.373
C01501=1203.361,305.598,-69.155,-176.524,7.336,148.373
C01502=1203.365,305.351,-69.124,-176.526,7.334,148.372
C01503=1203.369,305.103,-69.095,-176.529,7.331,148.372
C01504=1203.374,304.854,-69.065,-176.532,7.328,148.372
C01505=1203.378,304.606,-69.035,-176.534,7.325,148.372
C01506=1203.383,304.358,-69.005,-176.536,7.322,148.372
C01507=1203.387,304.110,-68.975,-176.538,7.320,148.373
C01508=1203.391,303.862,-68.945,-176.541,7.317,148.373
C01509=1203.396,303.613,-68.915,-176.544,7.314,148.373
C01510=1203.400,303.366,-68.885,-176.546,7.312,148.373
C01511=1203.404,303.117,-68.855,-176.549,7.309,148.373
C01512=1203.408,302.869,-68.826,-176.551,7.306,148.373
C01513=1203.413,302.621,-68.795,-176.554,7.304,148.373
C01514=1203.417,302.373,-68.766,-176.556,7.301,148.373
C01515=1203.421,302.125,-68.736,-176.558,7.298,148.373
C01516=1203.426,301.877,-68.706,-176.561,7.295,148.373
C01517=1203.430,301.628,-68.676,-176.564,7.292,148.373
C01518=1203.434,301.380,-68.647,-176.566,7.290,148.373
C01519=1203.438,301.132,-68.617,-176.569,7.287,148.373
C01520=1203.442,300.884,-68.588,-176.571,7.285,148.373
C01521=1203.447,300.636,-68.557,-176.573,7.282,148.373
C01522=1203.451,300.387,-68.527,-176.576,7.279,148.373
C01523=1203.455,300.139,-68.498,-176.578,7.277,148.373
C01524=1203.460,299.891,-68.469,-176.581,7.274,148.373
C01525=1203.464,299.642,-68.439,-176.583,7.272,148.373
C01526=1203.468,299.395,-68.408,-176.586,7.269,148.373
C01527=1203.473,299.146,-68.379,-176.588,7.266,148.373
C01528=1203.477,298.898,-68.349,-176.591,7.263,148.373
C01529=1203.481,298.650,-68.320,-176.593,7.260,148.373
C01530=1203.485,298.401,-68.291,-176.595,7.258,148.373
C01531=1203.489,298.153,-68.261,-176.598,7.255,148.373
C01532=1203.494,297.905,-68.231,-176.600,7.253,148.373
C01533=1203.498,297.656,-68.202,-176.603,7.250,148.373
C01534=1203.503,297.408,-68.172,-176.606,7.247,148.373
C01535=1203.507,297.160,-68.143,-176.608,7.245,148.373
C01536=1203.511,296.912,-68.113,-176.610,7.242,148.373
C01537=1203.516,296.664,-68.084,-176.613,7.239,148.374
C01538=1203.520,296.416,-68.055,-176.615,7.236,148.374
C01539=1203.524,296.167,-68.025,-176.618,7.233,148.374
C01540=1203.528,295.919,-67.996,-176.620,7.231,148.374
C01541=1203.532,295.671,-67.966,-176.623,7.228,148.374
C01542=1203.537,295.423,-67.937,-176.625,7.226,148.374
C01543=1203.541,295.174,-67.907,-176.628,7.223,148.374
C01544=1203.545,294.926,-67.878,-176.630,7.221,148.374
C01545=1203.549,294.678,-67.849,-176.633,7.218,148.374
C01546=1203.554,294.430,-67.819,-176.636,7.215,148.374
C01547=1203.558,294.182,-67.790,-176.638,7.213,148.374
C01548=1203.562,293.934,-67.761,-176.640,7.210,148.374
C01549=1203.566,293.685,-67.731,-176.642,7.208,148.374
C01550=1203.571,293.437,-67.702,-176.645,7.205,148.374
C01551=1203.575,293.188,-67.673,-176.647,7.202,148.374
C01552=1203.579,292.940,-67.643,-176.650,7.199,148.374
C01553=1203.584,292.692,-67.614,-176.652,7.197,148.374
C01554=1203.588,292.444,-67.585,-176.655,7.194,148.374
C01555=1203.592,292.196,-67.555,-176.658,7.192,148.375
C01556=1203.597,291.947,-67.527,-176.660,7.189,148.375
C01557=1203.601,291.699,-67.497,-176.663,7.186,148.375
C01558=1203.606,291.451,-67.468,-176.665,7.184,148.375
C01559=1203.610,291.203,-67.439,-176.668,7.181,148.375
C01560=1203.615,290.954,-67.410,-176.670,7.179,148.375
C01561=1203.619,290.706,-67.381,-176.672,7.176,148.375
C01562=1203.623,290.458,-67.351,-176.675,7.174,148.375
C01563=1203.627,290.210,-67.323,-176.678,7.171,148.375
C01564=1203.631,289.961,-67.294,-176.680,7.168,148.375
C01565=1203.636,289.713,-67.264,-176.683,7.166,148.375
C01566=1203.640,289.465,-67.235,-176.685,7.163,148.375
C01567=1203.645,289.190,-67.203,-176.688,7.160,148.375
C01568=1203.649,288.916,-67.172,-176.690,7.158,148.375
C01569=1203.655,288.641,-67.139,-176.693,7.155,148.376
C01570=1203.659,288.368,-67.107,-176.696,7.152,148.376
C01571=1203.664,288.119,-67.078,-176.699,7.149,148.376
C01572=1203.668,287.871,-67.049,-176.701,7.147,148.376
C01573=1203.672,287.623,-67.020,-176.704,7.144,148.376
C01574=1203.677,287.374,-66.992,-176.706,7.142,148.376
C01575=1203.681,287.126,-66.962,-176.709,7.139,148.376
C01576=1203.685,286.877,-66.933,-176.711,7.137,148.376
C01577=1203.689,286.630,-66.905,-176.714,7.134,148.376
C01578=1203.694,286.381,-66.876,-176.716,7.131,148.376
C01579=1203.698,286.133,-66.847,-176.719,7.129,148.377
C01580=1203.703,285.885,-66.818,-176.721,7.126,148.377
C01581=1203.707,285.637,-66.790,-176.724,7.123,148.377
C01582=1203.711,285.388,-66.761,-176.726,7.120,148.377
C01583=1203.715,285.140,-66.731,-176.729,7.118,148.377
C01584=1203.720,284.891,-66.703,-176.732,7.116,148.377
C01585=1203.724,284.643,-66.675,-176.734,7.113,148.377
C01586=1203.728,284.395,-66.645,-176.737,7.110,148.377
C01587=1203.733,284.146,-66.617,-176.739,7.108,148.377
C01588=1203.737,283.898,-66.588,-176.741,7.105,148.377
C01589=1203.741,283.649,-66.559,-176.744,7.103,148.377
C01590=1203.746,283.401,-66.531,-176.747,7.100,148.378
C01591=1203.750,283.153,-66.502,-176.749,7.098,148.378
C01592=1203.755,282.905,-66.474,-176.752,7.095,148.378
C01593=1203.759,282.656,-66.445,-176.754,7.093,148.378
C01594=1203.763,282.408,-66.416,-176.757,7.090,148.378
C01595=1203.768,282.160,-66.388,-176.759,7.088,148.378
C01596=1203.772,281.911,-66.359,-176.762,7.085,148.378
C01597=1203.776,281.663,-66.331,-176.764,7.083,148.378
C01598=1203.781,281.415,-66.302,-176.767,7.080,148.378
C01599=1203.785,281.167,-66.274,-176.769,7.078,148.378
C01600=1203.790,280.918,-66.245,-176.772,7.075,148.378
C01601=1203.794,280.669,-66.217,-176.774,7.073,148.379
C01602=1203.798,280.421,-66.188,-176.777,7.070,148.379
C01603=1203.803,280.173,-66.159,-176.779,7.068,148.379
C01604=1203.807,279.925,-66.131,-176.782,7.065,148.379
C01605=1203.812,279.677,-66.103,-176.784,7.063,148.379
C01606=1203.815,279.428,-66.075,-176.787,7.061,148.379
C01607=1203.820,279.180,-66.046,-176.789,7.058,148.379
C01608=1203.824,278.932,-66.017,-176.792,7.055,148.379
C01609=1203.828,278.683,-65.989,-176.794,7.052,148.379
C01610=1203.833,278.435,-65.961,-176.797,7.051,148.380
C01611=1203.837,278.186,-65.932,-176.800,7.048,148.380
C01612=1203.842,277.938,-65.904,-176.802,7.045,148.380
C01613=1203.846,277.689,-65.876,-176.804,7.042,148.380
C01614=1203.850,277.442,-65.848,-176.807,7.041,148.380
C01615=1203.855,277.193,-65.819,-176.810,7.038,148.380
C01616=1203.859,276.945,-65.791,-176.812,7.035,148.380
C01617=1203.864,276.696,-65.763,-176.815,7.033,148.380
C01618=1203.868,276.448,-65.735,-176.817,7.030,148.381
C01619=1203.873,276.199,-65.706,-176.820,7.027,148.381
C01620=1203.877,275.951,-65.678,-176.822,7.025,148.381
C01621=1203.881,275.703,-65.650,-176.825,7.023,148.381
C01622=1203.886,275.454,-65.622,-176.827,7.020,148.381
C01623=1203.890,275.206,-65.594,-176.829,7.018,148.381
C01624=1203.895,274.958,-65.565,-176.833,7.015,148.381
C01625=1203.898,274.709,-65.537,-176.835,7.013,148.381
C01626=1203.903,274.461,-65.509,-176.838,7.010,148.381
C01627=1203.907,274.212,-65.481,-176.840,7.008,148.382
C01628=1203.912,273.965,-65.453,-176.843,7.005,148.382
C01629=1203.915,273.716,-65.425,-176.845,7.003,148.382
C01630=1203.920,273.468,-65.396,-176.848,7.001,148.382
C01631=1203.924,273.219,-65.368,-176.850,6.998,148.382
C01632=1203.929,272.971,-65.341,-176.852,6.996,148.382
C01633=1203.933,272.722,-65.312,-176.856,6.993,148.382
C01634=1203.938,272.474,-65.285,-176.858,6.991,148.383
C01635=1203.941,272.225,-65.257,-176.860,6.988,148.383
C01636=1203.947,271.977,-65.228,-176.863,6.986,148.383
C01637=1203.951,271.729,-65.200,-176.866,6.983,148.383
C01638=1203.955,271.480,-65.173,-176.868,6.981,148.383
C01639=1203.960,271.232,-65.145,-176.870,6.979,148.383
C01640=1203.964,270.983,-65.116,-176.873,6.976,148.383
C01641=1203.968,270.735,-65.089,-176.875,6.974,148.383
C01642=1203.973,270.487,-65.062,-176.879,6.971,148.384
C01643=1203.977,270.238,-65.033,-176.881,6.969,148.384
C01644=1203.982,269.990,-65.005,-176.883,6.966,148.384
C01645=1203.986,269.741,-64.978,-176.886,6.964,148.384
C01646=1203.990,269.493,-64.950,-176.888,6.962,148.384
C01647=1203.995,269.245,-64.922,-176.891,6.959,148.384
C01648=1203.999,268.996,-64.894,-176.893,6.957,148.385
C01649=1204.003,268.748,-64.866,-176.896,6.954,148.385
C01650=1204.008,268.500,-64.839,-176.898,6.952,148.385
C01651=1204.012,268.251,-64.811,-176.901,6.950,148.385
C01652=1204.017,268.003,-64.783,-176.904,6.947,148.385
C01653=1204.021,267.754,-64.755,-176.906,6.945,148.385
C01654=1204.025,267.506,-64.728,-176.909,6.942,148.385
C01655=1204.030,267.258,-64.700,-176.911,6.940,148.385
C01656=1204.034,267.008,-64.672,-176.914,6.938,148.386
C01657=1204.038,266.761,-64.645,-176.916,6.935,148.386
C01658=1204.043,266.512,-64.618,-176.919,6.933,148.386
C01659=1204.048,266.264,-64.589,-176.922,6.930,148.386
C01660=1204.052,266.015,-64.562,-176.924,6.928,148.386
C01661=1204.056,265.767,-64.534,-176.926,6.926,148.386
C01662=1204.061,265.518,-64.507,-176.929,6.923,148.386
C01663=1204.065,265.270,-64.479,-176.931,6.921,148.387
C01664=1204.069,265.021,-64.452,-176.934,6.919,148.387
C01665=1204.074,264.773,-64.424,-176.937,6.916,148.387
C01666=1204.078,264.524,-64.396,-176.939,6.914,148.387
C01667=1204.082,264.276,-64.369,-176.942,6.911,148.387
C01668=1204.087,264.028,-64.342,-176.945,6.910,148.388
C01669=1204.091,263.780,-64.314,-176.947,6.907,148.388
C01670=1204.095,263.531,-64.286,-176.949,6.904,148.388
C01671=1204.100,263.258,-64.256,-176.952,6.903,148.388
C01672=1204.106,262.985,-64.226,-176.955,6.900,148.388
C01673=1204.110,262.712,-64.196,-176.958,6.897,148.388
C01674=1204.115,262.440,-64.165,-176.961,6.894,148.389
C01675=1204.120,262.191,-64.138,-176.963,6.892,148.389
C01676=1204.124,261.943,-64.111,-176.965,6.890,148.389
C01677=1204.128,261.694,-64.083,-176.969,6.887,148.389
C01678=1204.133,261.446,-64.056,-176.971,6.885,148.389
C01679=1204.137,261.197,-64.029,-176.973,6.883,148.389
C01680=1204.142,260.949,-64.002,-176.976,6.880,148.389
C01681=1204.146,260.701,-63.974,-176.979,6.878,148.390
C01682=1204.150,260.452,-63.947,-176.981,6.876,148.390
C01683=1204.155,260.203,-63.920,-176.984,6.873,148.390
C01684=1204.159,259.955,-63.893,-176.986,6.871,148.390
C01685=1204.163,259.707,-63.865,-176.988,6.869,148.390
C01686=1204.168,259.459,-63.838,-176.991,6.866,148.391
C01687=1204.172,259.209,-63.811,-176.994,6.864,148.391
C01688=1204.177,258.961,-63.784,-176.996,6.862,148.391
C01689=1204.181,258.712,-63.757,-176.999,6.859,148.391
C01690=1204.186,258.464,-63.730,-177.002,6.857,148.391
C01691=1204.190,258.216,-63.702,-177.004,6.855,148.391
C01692=1204.195,257.968,-63.675,-177.007,6.853,148.392
C01693=1204.198,257.719,-63.648,-177.009,6.850,148.392
C01694=1204.203,257.470,-63.621,-177.012,6.849,148.392
C01695=1204.208,257.222,-63.594,-177.014,6.845,148.392
C01696=1204.212,256.973,-63.567,-177.017,6.844,148.392
C01697=1204.217,256.725,-63.540,-177.019,6.841,148.392
C01698=1204.222,256.476,-63.513,-177.022,6.839,148.393
C01699=1204.225,256.228,-63.486,-177.024,6.837,148.393
C01700=1204.230,255.979,-63.459,-177.027,6.835,148.393
C01701=1204.234,255.730,-63.432,-177.030,6.832,148.393
C01702=1204.239,255.482,-63.405,-177.032,6.830,148.393
C01703=1204.244,255.233,-63.378,-177.035,6.828,148.394
C01704=1204.247,254.985,-63.351,-177.038,6.825,148.394
C01705=1204.252,254.737,-63.324,-177.040,6.823,148.394
C01706=1204.257,254.488,-63.297,-177.042,6.821,148.394
C01707=1204.261,254.240,-63.270,-177.045,6.818,148.394
C01708=1204.265,253.992,-63.244,-177.048,6.816,148.395
C01709=1204.269,253.742,-63.216,-177.050,6.814,148.395
C01710=1204.274,253.494,-63.189,-177.053,6.811,148.395
C01711=1204.278,253.246,-63.163,-177.055,6.809,148.395
C01712=1204.283,252.997,-63.136,-177.058,6.807,148.395
C01713=1204.287,252.749,-63.109,-177.060,6.805,148.395
C01714=1204.292,252.500,-63.081,-177.063,6.802,148.396
C01715=1204.296,252.252,-63.055,-177.065,6.800,148.396
C01716=1204.301,252.003,-63.029,-177.068,6.798,148.396
C01717=1204.305,251.754,-63.002,-177.071,6.795,148.396
C01718=1204.309,251.506,-62.975,-177.073,6.793,148.396
C01719=1204.314,251.258,-62.948,-177.075,6.791,148.397
C01720=1204.319,251.009,-62.921,-177.078,6.789,148.397
C01721=1204.323,250.760,-62.895,-177.081,6.786,148.397
C01722=1204.328,250.512,-62.868,-177.083,6.785,148.397
C01723=1204.331,250.264,-62.842,-177.086,6.782,148.397
C01724=1204.336,250.015,-62.815,-177.089,6.780,148.398
C01725=1204.341,249.767,-62.788,-177.091,6.778,148.398
C01726=1204.345,249.518,-62.762,-177.094,6.776,148.398
C01727=1204.350,249.269,-62.735,-177.096,6.774,148.398
C01728=1204.354,249.021,-62.708,-177.099,6.771,148.398
C01729=1204.359,248.772,-62.682,-177.102,6.769,148.399
C01730=1204.363,248.524,-62.655,-177.104,6.767,148.399
C01731=1204.367,248.275,-62.628,-177.106,6.765,148.399
C01732=1204.372,248.026,-62.602,-177.109,6.762,148.399
C01733=1204.376,247.778,-62.576,-177.112,6.760,148.399
C01734=1204.381,247.530,-62.549,-177.114,6.758,148.400
C01735=1204.385,247.281,-62.523,-177.117,6.755,148.400
C01736=1204.390,247.032,-62.496,-177.120,6.753,148.400
C01737=1204.393,246.784,-62.469,-177.122,6.751,148.400
C01738=1204.398,246.535,-62.443,-177.124,6.749,148.401
C01739=1204.402,246.287,-62.416,-177.127,6.746,148.401
C01740=1204.407,246.038,-62.390,-177.130,6.745,148.401
C01741=1204.411,245.790,-62.364,-177.132,6.742,148.401
C01742=1204.416,245.540,-62.337,-177.134,6.741,148.401
C01743=1204.420,245.292,-62.311,-177.138,6.738,148.402
C01744=1204.426,245.044,-62.285,-177.140,6.736,148.402
C01745=1204.430,244.796,-62.258,-177.142,6.734,148.402
C01746=1204.435,244.547,-62.232,-177.145,6.732,148.402
C01747=1204.438,244.298,-62.206,-177.148,6.729,148.402
C01748=1204.443,244.049,-62.179,-177.150,6.727,148.403
C01749=1204.447,243.801,-62.153,-177.153,6.725,148.403
C01750=1204.452,243.552,-62.127,-177.155,6.723,148.403
C01751=1204.456,243.304,-62.100,-177.157,6.721,148.403
C01752=1204.460,243.055,-62.074,-177.161,6.718,148.403
C01753=1204.465,242.806,-62.047,-177.163,6.716,148.404
C01754=1204.470,242.558,-62.022,-177.165,6.714,148.404
C01755=1204.474,242.310,-61.996,-177.168,6.712,148.404
C01756=1204.479,242.061,-61.969,-177.171,6.709,148.404
C01757=1204.483,241.812,-61.943,-177.173,6.708,148.405
C01758=1204.487,241.564,-61.917,-177.176,6.706,148.405
C01759=1204.492,241.315,-61.890,-177.178,6.703,148.405
C01760=1204.496,241.066,-61.865,-177.181,6.701,148.405
C01761=1204.501,240.819,-61.839,-177.184,6.699,148.406
C01762=1204.506,240.570,-61.812,-177.186,6.697,148.406
C01763=1204.510,240.321,-61.786,-177.189,6.695,148.406
C01764=1204.514,240.073,-61.760,-177.191,6.693,148.406
C01765=1204.519,239.823,-61.734,-177.194,6.690,148.406
C01766=1204.523,239.575,-61.708,-177.197,6.688,148.407
C01767=1204.528,239.327,-61.683,-177.199,6.686,148.407
C01768=1204.532,239.078,-61.655,-177.201,6.684,148.407
C01769=1204.537,238.829,-61.630,-177.204,6.682,148.407
C01770=1204.541,238.580,-61.604,-177.207,6.679,148.407
C01771=1204.545,238.332,-61.578,-177.209,6.678,148.408
C01772=1204.551,238.083,-61.552,-177.212,6.676,148.408
C01773=1204.555,237.835,-61.526,-177.214,6.674,148.408
C01774=1204.559,237.586,-61.500,-177.217,6.672,148.409
C01775=1204.564,237.314,-61.472,-177.220,6.669,148.409
C01776=1204.569,237.044,-61.444,-177.222,6.667,148.409
C01777=1204.574,236.772,-61.415,-177.225,6.664,148.409
C01778=1204.579,236.500,-61.387,-177.228,6.662,148.410
C01779=1204.583,236.252,-61.361,-177.231,6.660,148.410
C01780=1204.587,236.003,-61.335,-177.233,6.657,148.410
C01781=1204.592,235.755,-61.309,-177.236,6.656,148.410
C01782=1204.596,235.506,-61.284,-177.239,6.654,148.411
C01783=1204.601,235.257,-61.258,-177.241,6.652,148.411
C01784=1204.606,235.009,-61.232,-177.243,6.650,148.411
C01785=1204.610,234.760,-61.206,-177.247,6.647,148.411
C01786=1204.615,234.512,-61.181,-177.249,6.645,148.411
C01787=1204.619,234.263,-61.155,-177.251,6.643,148.412
C01788=1204.623,234.014,-61.129,-177.254,6.641,148.412
C01789=1204.627,233.765,-61.103,-177.256,6.639,148.412
C01790=1204.633,233.517,-61.077,-177.259,6.636,148.412
C01791=1204.637,233.268,-61.052,-177.262,6.635,148.413
C01792=1204.641,233.019,-61.026,-177.265,6.633,148.413
C01793=1204.646,232.771,-61.001,-177.267,6.631,148.413
C01794=1204.650,232.522,-60.975,-177.269,6.629,148.413
C01795=1204.655,232.273,-60.949,-177.272,6.627,148.414
C01796=1204.659,232.025,-60.924,-177.275,6.624,148.414
C01797=1204.664,231.777,-60.898,-177.277,6.622,148.414
C01798=1204.668,231.528,-60.872,-177.280,6.620,148.414
C01799=1204.673,231.279,-60.847,-177.282,6.618,148.415
C01800=1204.677,231.030,-60.822,-177.285,6.616,148.415
C01801=1204.682,230.781,-60.796,-177.287,6.614,148.415
C01802=1204.686,230.533,-60.771,-177.290,6.612,148.416
C01803=1204.691,230.285,-60.745,-177.293,6.609,148.416
C01804=1204.695,230.036,-60.719,-177.295,6.608,148.416
C01805=1204.700,229.788,-60.694,-177.298,6.606,148.416
C01806=1204.704,229.538,-60.669,-177.300,6.604,148.416
C01807=1204.709,229.290,-60.643,-177.303,6.602,148.417
C01808=1204.713,229.041,-60.618,-177.305,6.600,148.417
C01809=1204.717,228.792,-60.592,-177.309,6.597,148.417
